(* IEC 61131-3 sources: elnaProjects/ElpcLogic/PomarKc7Unchanged/build_USO_ecl (part 4) *)

  IF getSdvig THEN StrSw.sdvig:= TRUE; END_IF;

  sdvigReset(IN:=StrSw.sdvig, PT:=T#15S);

  IF sdvigReset.Q THEN StrSw.sdvig:=FALSE; END_IF;

  lastOnStatus := StrSw.onStatus;

  (* ---- Распаковка команды ---- *)
  _sunpackerCommand(command := StrSw.inCommand);
  	cmd := _sunpackerCommand.cmd;
  	source := _sunpackerCommand.source;

  (* ---- Обработка команды ---- *)
  IF cmd <> 0 AND lastCmd <> cmd and (((NOT StrSw.opcCommandsDisabled) AND source > 0) OR source = 0) then
  	CASE BYTE_TO_INT(cmd) OF
  	(*cmd_open*) 1 :
  			IF  StrSw.ISVALIDREF_cmdOn THEN StrSw.CmdOn := TRUE;
  				IF StrSw.ISVALIDREF_cmdOff THEN StrSw.CmdOff := FALSE; END_IF;
  			ELSIF  StrSw.ISVALIDREF_cmdOff THEN StrSw.CmdOff := FALSE;  END_IF;
                                lastCmd := cmd;
  			errorCMDTimer(IN := false);
  			_commandErrorTimer := true;
  			StrSw.lastCmdIsOn := true;
  	(*cmd_close*) 2 :
  			IF StrSw.ISVALIDREF_cmdOff THEN StrSw.CmdOff := TRUE;
  				IF StrSw.ISVALIDREF_cmdOn THEN StrSw.CmdOn := FALSE; END_IF;
  			ELSIF StrSw.ISVALIDREF_cmdOn THEN StrSw.CmdOn := FALSE; END_IF;
                                lastCmd := cmd;
  			errorCMDTimer(IN := false);
  			_commandErrorTimer := true;
  			StrSw.lastCmdIsOn := false;
  	(*cmd_reset*) 3 :    IF StrSw.ISVALIDREF_statOn OR StrSw.ISVALIDREF_statOff THEN
  			StrSw.CmdOn := FALSE;
  			StrSw.CmdOff := FALSE;
                                lastCmd :=0;
  			_commandErrorTimer := false;
  			StrSw.lastCmdIsOn := false;
                                 END_IF;
  	END_CASE;
  	source_for_Status := source;
  	cmd_for_Status := cmd;
  	command_error_for_Status := 0;
  END_IF;

  errorCMDTimer(In := _commandErrorTimer, PT :=T#10s);

  (* ---- алгоритм  для команды ВКЛючить ---- *)
  IF (StrSw.onStatus = _statusDualInput.STATUS_ON) and StrSw.lastCmdIsOn then
  	IF StrSw.ISVALIDREF_cmdOn AND StrSw.ISVALIDREF_cmdOff then  StrSw.cmdOn := false; END_IF;

  	 errorCMDTimer(In := false);
  	 _commandErrorTimer := false;
  	 cmd_for_Status := 0;
  	 source_for_Status := 0;
  END_IF;

  (* ---- off ---- *)
  IF (StrSw.onStatus = _statusDualInput.STATUS_OFF) and (NOT StrSw.lastCmdIsOn) then
  	IF StrSw.ISVALIDREF_cmdOn AND StrSw.ISVALIDREF_cmdOff then  StrSw.cmdOff := false; END_IF;

  	 errorCMDTimer(In := false);
  	 _commandErrorTimer := false;
  	 cmd_for_Status := 0;
  	 source_for_Status := 0;
  END_IF;

  (* ---- ошибка исполнения команды ---- *)
  if errorCMDTimer.Q and (cmd_for_Status <> 0) then
  	command_error_for_Status :=  cmd_for_Status;
  	_commandErrorTimer := false;
  	StrSw.CmdOn := false;
  	StrSw.CmdOff := false;
  	lastCmd := 0;
  end_if;

  (* ---- сброс ошибки команды ---- *)
  StrSw.CommandFault := command_error_for_Status <> 0;
  _errorReset(IN := command_error_for_Status <> 0, PT := T#5S);
  IF _errorReset.Q THEN
  	cmd_for_Status := 0;
  	source_for_Status := 0;
  	command_error_for_Status := 0;
  END_IF;

  outputsSets(in := (StrSw.ISVALIDREF_cmdOn and StrSw.cmdOn ) OR (StrSw.ISVALIDREF_cmdOff and StrSw.cmdOff), PT := T#2S);
  	IF NOT outputsSets.Q THEN
  		StrSw.BreakCmdOn := inBreakCmdOn._inversed AND
                      inBreakCmdOn.reliability AND StrSw.ISVALIDREF_inBreakCmdOn;

  		StrSw.BreakCmdOff := inBreakCmdOff._inversed
                      AND inBreakCmdOff.reliability AND StrSw.ISVALIDREF_inBreakCmdOff;
  	END_IF;

  cmdOn := StrSw.cmdOn;
  cmdOff:= StrSw.cmdOff;

  (* ---- формирование зашифрованного статуса для АРМа ---- *)
  StrSw.status := shl(BYTE_TO_DWORD(source_for_Status), 29)
  		OR shl(BYTE_TO_DWORD(cmd_for_Status), 26)
  		OR shl(BYTE_TO_DWORD(command_error_for_Status), 23)
  		OR shl(bool_to_DWORD(StrSw.sdvig), 22)
  		OR shl(bool_to_DWORD(StrSw.OpcCommandsDisabled), 21)
                      OR shl(bool_to_DWORD(StrSw.lastCmdIsOn), 14)
                      OR shl(BOOL_TO_DWORD(StrSw.BreakCmdOff), 13)
  		OR shl(BOOL_TO_DWORD(StrSw.BreakCmdOn), 12)
  		OR shl(BOOL_TO_DWORD(StrSw.ErrorBlock), 11)
  		OR shl(BOOL_TO_DWORD(StrSw.ErrorPowerOff), 10)
  		OR shl(BOOL_TO_DWORD(StrSw.Manual), 8)
  		OR shl(BOOL_TO_DWORD(StrSw.Auto), 7)
  		OR shl(BOOL_TO_DWORD(StrSw.Distance), 6)
  		OR shl(BOOL_TO_DWORD(StrSw.Local), 5)
  		OR shl(BOOL_TO_DWORD(StrSw.Ns), 4)
                  	OR shl(BOOL_TO_DWORD(StrSw.Accident ),3)
  		OR BYTE_TO_DWORD(StrSw.onStatus);
END_FUNCTION_BLOCK

FUNCTION_BLOCK fb_SectionSwitch
  VAR_INPUT
    statOn : BOOL;
    statOff : BOOL;
    statOn_reliability : BOOL;
    statOff_reliability : BOOL;
  END_VAR
  VAR_IN_OUT
    StrSw : struct_SectionSwitch;
  END_VAR
  VAR_INPUT
    basketRolledIn : TYPE_ReliableBit;
    basketRolledOut : TYPE_ReliableBit;
    basketTest : TYPE_ReliableBit;
    inNs : TYPE_ReliableBit;
    inoffKNA : TYPE_ReliableBit;
    inAccident : TYPE_ReliableBit;
    inLocal : TYPE_ReliableBit;
    inDistance : TYPE_ReliableBit;
    inBreakCmdOn : TYPE_ReliableBit;
    inBreakCmdOff : TYPE_ReliableBit;
  END_VAR
  VAR
    onInit : BOOL := FALSE;
    _statOn : BOOL;
    _statOff : BOOL;
    getSdvig : BOOL;
    lastOnStatus : BYTE;
    cmd : BYTE;
    source : BYTE;
    lastCmd : BYTE;
    source_for_Status : BYTE;
    cmd_for_Status : BYTE;
    command_error_for_Status : BYTE;
    _basketRolledIn : TYPE_ReliableBit;
    _basketRolledOut : TYPE_ReliableBit;
    _basketTest : TYPE_ReliableBit;
    _sunpackerCommand : fb_sunpackerCommand;
    _statusDualInput : TYPE_statusDualInput;
    _statusBasket : TYPE_basketStats;
    _commandDualInput : TYPE_commandDualInput;
    _commandErrorTimer : BOOL;
    resetErrorTimer : BOOL;
    _changWithoutCommand : BOOL;
    errorCMDTimer : TON;
    _errorReset : TON;
    sdvigReset : TON;
    outputsSets : TOF;
  END_VAR
  VAR_IN_OUT
    cmdOn : BOOL;
    cmdOff : BOOL;
  END_VAR

  IF NOT onInit THEN
  IF StrSw.ISVALIDREF_cmdOn XOR StrSw.ISVALIDREF_cmdOff THEN
  	IF 	StrSw.ISVALIDREF_cmdOn THEN
  		lastCmd:= 2; (*baseCmdOff*)
  	ELSE
  		lastCmd:= 1; (*baseCmdOn*)
  	END_IF;
  END_IF;
  onInit:=TRUE;
  END_IF;

  (* ---- Формирование состояния тележки ---- *)

  IF (NOT StrSw.ISVALIDREF_basketRolledIn) AND (NOT StrSw.ISVALIDREF_basketRolledOut) THEN
            StrSw.basketStatus:=_statusBasket.BASKET_NOTDEFINED;
  ELSE
  		IF StrSw.ISVALIDREF_basketTest THEN
  		_basketTest:=basketTest;
  	ELSE
  		_basketTest.reliability:=TRUE;
  		_basketTest.value :=FALSE;
  	END_IF;

  	IF StrSw.ISVALIDREF_basketRolledIn THEN
  		_basketRolledIn:=basketRolledIn;
  	ELSE
  		_basketRolledIn:=basketRolledOut;
  		IF StrSw.ISVALIDREF_basketTest THEN
  		_basketRolledIn.value:=NOT (_basketRolledIn.value OR _basketTest.value);
  		ELSE
  		_basketRolledIn.value:= NOT _basketRolledIn.value;
  		END_IF;

  	END_IF;

  	IF StrSw.ISVALIDREF_basketRolledOut THEN
  		_basketRolledOut:=basketRolledOut;
  	ELSE
  		_basketRolledOut:=basketRolledIn;
  		IF StrSw.ISVALIDREF_basketTest THEN
  		_basketRolledOut.value:= NOT (_basketRolledOut.value OR _basketTest.value );
  		ELSE
  			_basketRolledOut.value := NOT _basketRolledout.value;
  		END_IF;

  	END_IF;

  IF _basketRolledIn.reliability AND _basketRolledOut.reliability AND _basketTest.reliability THEN
  		IF (BOOL_TO_INT(_basketRolledIn.value)+BOOL_TO_INT(_basketRolledOut.value)+BOOL_TO_INT(_basketTest.value))=1 THEN
  			IF _basketRolledIn.value THEN
  				StrSw.basketStatus:=_statusBasket.BASKET_ROLLEDIN;
  			ELSIF _basketRolledOut.value THEN
  				StrSw.basketStatus:=_statusBasket.BASKET_ROLLEDOUT;
  			ELSIF _basketTest.value THEN
  				StrSw.basketStatus:=_statusBasket.BASKET_TEST;
  			END_IF;
  		ELSE
  			StrSw.basketStatus:=_statusBasket.BASKET_ERROR;
  		END_IF;
  	ELSE
  		StrSw.basketStatus:=_statusBasket.BASKET_NOTDEFINED;
  	END_IF;
  END_IF;

  (* ---- Если управление с ВУ заблокировано, то в ИМ передаем команду из алгоритма ---- *)
  IF StrSw.inOpcCommandsDisabled THEN
  	StrSw.inCommand := StrSw.inCommand_Alg;
  ELSE (* иначе передаем команду с АРМа*)
  	StrSw.inCommand := StrSw.inCommand_ARM;
  END_IF;

  (* ---- Формирование состояния механизма ---- *)

  IF (StrSw.ISVALIDREF_statOn) OR (StrSw.ISVALIDREF_statOff) THEN
  	IF (StrSw.ISVALIDREF_statOn) AND (StrSw.ISVALIDREF_statOff) THEN
  	StrSw.reliability:= statOn_reliability AND statOff_reliability;
  		_statOn  := statOn;
  		_statOff := statOff;
  	ELSIF (StrSw.ISVALIDREF_statOn) THEN
                       StrSw.reliability:= statOn_reliability;
  		_statOn  := statOn;
  		_statOff := NOT statOn;
  	ELSIF (StrSw.ISVALIDREF_statOff) THEN
  		 StrSw.reliability:= statOff_reliability;
  		_statOn  := NOT statOff;
  		_statOff :=statOff;
  	END_IF;

  	IF StrSw.reliability THEN
  		IF _statOn AND NOT _statOff 		THEN 	StrSw.onStatus := _statusDualInput.STATUS_ON;
  		ELSIF _statOff AND NOT _statOn 	THEN 	StrSw.onStatus := _statusDualInput.Status_OFF;
  		ELSIF NOT _statOn AND NOT _statOff 	THEN 	StrSw.onStatus := _statusDualInput.STATUS_TRANSITIONAL;
  		ELSE					StrSw.onStatus := _statusDualInput.STATUS_ERROR;
                      END_IF;

  	ELSE
  		StrSw.onStatus := _statusDualInput.STATUS_NOTDEFINED;

  	END_IF;
  ELSE
  	CASE BYTE_TO_INT(lastCmd) OF
  		(*baseCmdOn*) 1: StrSw.onStatus  := _statusDualInput.STATUS_ON;
  		(*baseCmdOff*) 2: StrSw.onStatus  := _statusDualInput.STATUS_OFF;

  	ELSE
  		 StrSw.onStatus := _statusDualInput.STATUS_NOTDEFINED;

  	END_CASE;
  END_IF;

  StrSw.Accident := inAccident.value AND inAccident.reliability;
  StrSw.Ns := inNs.value AND inNs.reliability;
  StrSw.Local := inLocal.value AND inLocal.reliability;
  StrSw.Distance := inDistance.value AND inDistance.reliability;
  StrSw.OpcCommandsDisabled := StrSw.inOpcCommandsDisabled;
  StrSw.offKNA := inoffKNA.value AND inoffKNA.reliability;

  (* ---- Формирование признака сдвига ---- *)

  getSdvig := FALSE;
  IF (StrSw.ISVALIDREF_cmdOn OR StrSw.ISVALIDREF_cmdOff) AND NOT StrSw.Local THEN
  	IF NOT (StrSw.CmdOn OR StrSw.CmdOff) THEN
                       IF (lastOnStatus <> StrSw.onStatus AND
  		(StrSw.onStatus <> _statusDualInput.STATUS_NOTDEFINED AND
                       StrSw.onStatus <> _statusDualInput.STATUS_ERROR)     AND
  		(lastOnStatus <> _statusDualInput.STATUS_NOTDEFINED   AND
                       lastOnStatus <> _statusDualInput.STATUS_ERROR))
                      THEN
  			getSdvig   := TRUE;
  		END_IF;
  	END_IF;
  END_IF;

  IF getSdvig THEN StrSw.sdvig:= TRUE; END_IF;

  sdvigReset(IN:=StrSw.sdvig, PT:=T#15S);

  IF sdvigReset.Q THEN StrSw.sdvig:=FALSE; END_IF;

  lastOnStatus := StrSw.onStatus;

  (* ---- Распаковка команды ---- *)
  _sunpackerCommand(command := StrSw.inCommand);
  	cmd := _sunpackerCommand.cmd;
  	source := _sunpackerCommand.source;

  (* ---- Обработка команды ---- *)
  IF cmd <> 0 AND lastCmd <> cmd and (((NOT StrSw.opcCommandsDisabled) AND source > 0) OR source = 0) then
  	CASE BYTE_TO_INT(cmd) OF
  	(*cmd_open*) 1 :
  			IF  StrSw.ISVALIDREF_cmdOn THEN StrSw.CmdOn := TRUE;
  				IF StrSw.ISVALIDREF_cmdOff THEN StrSw.CmdOff := FALSE; END_IF;
  			ELSIF  StrSw.ISVALIDREF_cmdOff THEN StrSw.CmdOff := FALSE;  END_IF;
  			errorCMDTimer(IN := false);
  			_commandErrorTimer := true;
  			StrSw.lastCmdIsOn := true;
  	(*cmd_close*) 2 :
  			IF StrSw.ISVALIDREF_cmdOff THEN StrSw.CmdOff := TRUE;
  				IF StrSw.ISVALIDREF_cmdOn THEN StrSw.CmdOn := FALSE; END_IF;
  			ELSIF StrSw.ISVALIDREF_cmdOn THEN StrSw.CmdOn := FALSE; END_IF;
  			errorCMDTimer(IN := false);
  			_commandErrorTimer := true;
  			StrSw.lastCmdIsOn := false;
  	(*cmd_reset*) 3 :    IF StrSw.ISVALIDREF_statOn OR StrSw.ISVALIDREF_statOff THEN
  			StrSw.CmdOn := FALSE;
  			StrSw.CmdOff := FALSE;
                                lastCmd := 0;
  			_commandErrorTimer := false;
  			StrSw.lastCmdIsOn := false;
                                 END_IF;
  	END_CASE;
  	source_for_Status := source;
  	cmd_for_Status := cmd;
  	command_error_for_Status := 0;
  END_IF;
  lastCmd := cmd;

  errorCMDTimer(In := _commandErrorTimer, PT :=T#10s);

  (* ---- алгоритм  для команды ВКЛючить ---- *)
  IF (StrSw.onStatus = _statusDualInput.STATUS_ON) and (StrSw.lastCmdIsOn) then
  	IF StrSw.ISVALIDREF_cmdOn AND StrSw.ISVALIDREF_cmdOff then  StrSw.cmdOn := false; END_IF;

  	 errorCMDTimer(In := false);
  	 _commandErrorTimer := false;
  	 cmd_for_Status := 0;
  	 source_for_Status := 0;
  END_IF;

  (* ---- off ---- *)
  IF (StrSw.onStatus = _statusDualInput.STATUS_OFF) and (NOT StrSw.lastCmdIsOn) then
  	IF StrSw.ISVALIDREF_cmdOn AND StrSw.ISVALIDREF_cmdOff then  StrSw.cmdOff := false; END_IF;

  	 errorCMDTimer(In := false);
  	 _commandErrorTimer := false;
  	 cmd_for_Status := 0;
  	 source_for_Status := 0;
  END_IF;

  (* ---- ошибка исполнения команды ---- *)
  if errorCMDTimer.Q and (cmd_for_Status <> 0) then
  	command_error_for_Status :=  cmd_for_Status;
  	_commandErrorTimer := false;
  	StrSw.CmdOn := false;
  	StrSw.CmdOff := false;
  	lastCmd := 0;
  end_if;

  (* ---- сброс ошибки команды ---- *)
  StrSw.CommandFault := command_error_for_Status <> 0;
  _errorReset(IN := command_error_for_Status <> 0, PT := T#5S);
  IF _errorReset.Q THEN
  	cmd_for_Status := 0;
  	source_for_Status := 0;
  	command_error_for_Status := 0;
  END_IF;

  outputsSets(in := (StrSw.ISVALIDREF_cmdOn and StrSw.cmdOn ) OR (StrSw.ISVALIDREF_cmdOff and StrSw.cmdOff), PT := T#2S);
  	IF NOT outputsSets.Q THEN
  		StrSw.BreakCmdOn := inBreakCmdOn._inversed AND inBreakCmdOn.reliability AND StrSw.ISVALIDREF_inBreakCmdOn;
  		StrSw.BreakCmdOff := inBreakCmdOff._inversed AND inBreakCmdOff.reliability AND StrSw.ISVALIDREF_inBreakCmdOff;
  	END_IF;

  cmdOn := StrSw.cmdOn;
  cmdOff:= StrSw.cmdOff;

  (* ---- формирование зашифрованного статуса для АРМа ---- *)
  StrSw.status := shl(BYTE_TO_DWORD(source_for_Status), 29)
  		OR shl(BYTE_TO_DWORD(cmd_for_Status), 26)
  		OR shl(BYTE_TO_DWORD(command_error_for_Status), 23)
  		OR shl(bool_to_DWORD(StrSw.sdvig), 22)
  		OR shl(bool_to_DWORD(StrSw.OpcCommandsDisabled), 21)
                      OR shl(BOOL_TO_DWORD(StrSw.offKNA), 17)
                      OR shl(bool_to_DWORD(StrSw.lastCmdIsOn), 14)
                      OR shl(BOOL_TO_DWORD(StrSw.BreakCmdOff), 13)
  		OR shl(BOOL_TO_DWORD(StrSw.BreakCmdOn), 12)
                      OR shl(BYTE_TO_DWORD(StrSw.basketStatus), 8)
  		OR shl(BOOL_TO_DWORD(StrSw.Distance), 6)
  		OR shl(BOOL_TO_DWORD(StrSw.Local), 5)
  		OR shl(BOOL_TO_DWORD(StrSw.Ns), 4)
                  	OR shl(BOOL_TO_DWORD(StrSw.Accident ),3)
  		OR BYTE_TO_DWORD(StrSw.onStatus);
END_FUNCTION_BLOCK

FUNCTION_BLOCK fb_meandr
  VAR
    _output : BOOL;
  END_VAR
  VAR_INPUT
    period : TIME := T#300MS;
  END_VAR
  VAR
    timer : TON;
    FALSE_val : BOOL := FALSE;
    TRUE_val : BOOL := TRUE;
  END_VAR
  VAR_IN_OUT
    output : BOOL;
  END_VAR

  timer(in:=NOT FALSE_val,PT:=period);

  IF timer.Q THEN
      _output:=_output XOR TRUE_val;
      timer(in:=FALSE);
  END_IF;

  output:=_output;
END_FUNCTION_BLOCK

FUNCTION_BLOCK fb_singleSignal
  VAR_INPUT
    signal : TYPE_ReliableBit;
  END_VAR
  VAR_IN_OUT
    str_SS : struct_singleSignal;
  END_VAR
  VAR
    TimerOn : TON;
    TimerOff : TOF;
  END_VAR

  str_SS.reliability:=signal.reliability;

  IF NOT str_SS.inverse THEN
  TimerOn(IN:=(signal.value AND str_SS.reliability AND NOT str_SS.Disabled_Sig), PT:=str_SS.DelayOn);
  ELSE
  TimerOn(IN:=(signal._inversed AND str_SS.reliability AND NOT str_SS.Disabled_Sig), PT:=str_SS.DelayOn);
  END_IF;

  TimerOff(IN:=TimerOn.Q, PT:=str_SS.DelayOff);

  str_SS.Q:=TimerOff.Q;

  str_SS.status:= SHL(BOOL_TO_DWORD(NOT str_SS.reliability), 15)
  	OR BOOL_TO_DWORD(str_SS.Q);
END_FUNCTION_BLOCK

FUNCTION_BLOCK fb_singleOutput
  VAR_IN_OUT
    signal : BOOL;
    str_SO : struct_singleOutput;
  END_VAR
  VAR
    pulseTimer : TON;
    resetCmdTimer : TON;
    TON_Command : TON;
    source : BYTE;
    cmd : BYTE;
    lastCmd : BYTE;
    source_for_Status : BYTE;
    cmd_for_Status : BYTE;
    command_error_for_Status : BYTE;
    pulseTimerPriznak : BOOL;
    resetCmdTimerPriznak : BOOL;
    _sunpackerCommand : fb_sunpackerCommand;
  END_VAR

  str_SO.OpcCommandsDisabled := str_SO.inOpcCommandsDisabled;

  (* ---- Если управление с ВУ заблокировано, то передаем команду из алгоритма ---- *)
  IF str_SO.inOpcCommandsDisabled THEN
  	str_SO.inCommand := str_SO.inCommand_Alg;
  ELSE (* иначе передаем команду с АРМа*)
  	str_SO.inCommand := str_SO.inCommand_ARM;
  END_IF;

  (*Распаковка команды*)
  _sunpackerCommand(command := str_SO.inCommand);
  	cmd := _sunpackerCommand.cmd;
  	source := _sunpackerCommand.source;

  (*Обработка команды*)
  IF cmd <> 0 AND lastCmd <> cmd and (((NOT str_SO.OpcCommandsDisabled) AND source > 0) OR source = 0) then
  	CASE BYTE_TO_INT(cmd) OF
  	(*cmd_on*) 1 :
  			str_SO.Q := TRUE;
  			pulseTimer(IN := FALSE);
  			pulseTimerPriznak := FALSE;
  			resetCmdTimer(IN := FALSE);
  			resetCmdTimerPriznak := TRUE;
  	(*cmd_off*) 2 :
  			str_SO.Q := FALSE;
  			pulseTimer(IN := FALSE);
  			pulseTimerPriznak := FALSE;
  			resetCmdTimer(IN := FALSE);
  			resetCmdTimerPriznak := TRUE;
  	(*cmd_pulse*) 3 :
  			str_SO.Q := TRUE;
                                pulseTimer(IN := FALSE);
                                pulseTimerPriznak := TRUE;
  			resetCmdTimer(IN := FALSE);
                                resetCmdTimerPriznak := FALSE;
  	END_CASE;
  	source_for_Status := source;
  	cmd_for_Status := cmd;
  	command_error_for_Status := 0;
  END_IF;
  lastCmd := cmd;

  pulseTimer(IN := pulseTimerPriznak, PT := str_SO.wait_time);
  pulseTimer();
  IF pulseTimer.Q THEN
  	pulseTimer(IN := FALSE);
  	pulseTimerPriznak := FALSE;

  	str_SO.Q := FALSE;

  	source_for_Status := 0;
  	cmd_for_Status := 0;
  	command_error_for_Status := 0;
  END_IF;

  resetCmdTimer(IN := resetCmdTimerPriznak, PT := T#10S);
  resetCmdTimer();
  IF resetCmdTimer.Q THEN
  	resetCmdTimer(IN := FALSE);
  	resetCmdTimerPriznak := FALSE;

  	source_for_Status := 0;
  	cmd_for_Status := 0;
  	command_error_for_Status := 0;
  END_IF;

  signal:= str_SO.Q;

  (*TON_Command(IN:= (inCommand <> 0) AND (source = 0), PT:= T#2S);*)
      (*IF TON_Command.Q THEN*)
          (*inCommand := 0;*)
      (*END_IF;*)
  str_SO.status :=                           shl(BYTE_TO_DWORD(source_for_Status), 29)
  				OR shl(BYTE_TO_DWORD(cmd_for_Status), 26)
  				OR shl(BYTE_TO_DWORD(command_error_for_Status), 23)
  				OR shl(BOOL_TO_DWORD(str_SO.OpcCommandsDisabled), 21)
  				OR BOOL_TO_DWORD(str_SO.Q);
END_FUNCTION_BLOCK

FUNCTION_BLOCK fb_DiscretParametr
  VAR_IN_OUT
    StrDP : struct_DiscretParametr;
  END_VAR
  VAR
    _sunpackerCommand : fb_sunpackerCommand;
    source : BYTE;
    cmd : BYTE;
    parametr : BYTE;
    lastParametr : BYTE;
    source_for_Status : BYTE;
    cmd_for_Status : BYTE;
    command_error_for_Status : BYTE;
    resetCmdTimer : TON;
    resetCmdTimerPriznak : BOOL;
    secondTact : BOOL;
  END_VAR

  IF NOT secondTact THEN
  	StrDP.Value := StrDP.currentValue;
  	secondTact := true;
  END_IF;

  StrDP.OpcCommandsDisabled := StrDP.inOpcCommandsDisabled;

  (* ---- Если управление с ВУ заблокировано, то передаем команду из алгоритма ---- *)
  IF StrDP.inOpcCommandsDisabled THEN
  	StrDP.inCommand := StrDP.inCommand_Alg;
  ELSE (* иначе передаем команду с АРМа*)
  	StrDP.inCommand := StrDP.inCommand_ARM;
  END_IF;

  _sunpackerCommand(command := StrDP.inCommand);
  	source := _sunpackerCommand.source;
            parametr := _sunpackerCommand.parametr;
  	cmd := _sunpackerCommand.cmd;

  IF NOT StrDP.inOpcCommandsDisabled THEN
  StrDP.newValue:= BYTE_TO_UINT(parametr);
  END_IF;

  IF cmd <> 0 AND StrDP.Value <> StrDP.newValue AND (((NOT StrDP.opcCommandsDisabled) AND source > 0) OR source = 0) then
  	CASE BYTE_TO_INT(cmd) OF
  	(*cmd_ChangeValue*) 1 :
                                    StrDP.Value := StrDP.newValue;
                                    StrDP.opcCommandsDisabled:=FALSE;
  	END_CASE;
  	source_for_Status := source;
  	cmd_for_Status := cmd;
  	resetCmdTimer(IN := FALSE);
  	resetCmdTimerPriznak := TRUE;
  END_IF;

  lastParametr := parametr;

  StrDP.status := SHL(BYTE_TO_DWORD(source_for_Status), 29)
  			OR SHL(BYTE_TO_DWORD(cmd_for_Status), 26)
  			OR SHL(BYTE_TO_DWORD(command_error_for_Status), 23)
  			OR SHL(BOOL_TO_DWORD(StrDP.OpcCommandsDisabled ), 21)
                                OR SHL(UINT_TO_DWORD(StrDP.Value), 5);

  resetCmdTimer(IN := resetCmdTimerPriznak, PT := T#5S);
  IF resetCmdTimer.Q THEN
  	resetCmdTimerPriznak := FALSE;
  	source_for_Status := 0;
  	cmd_for_Status := 0;
  	command_error_for_Status := 0;
  END_IF;
END_FUNCTION_BLOCK

FUNCTION_BLOCK fb_AnalogParametr
  VAR_IN_OUT
    StrAP : struct_AnalogParametr;
  END_VAR
  VAR
    _sunpackerCommand : fb_sunpackerCommand;
    source : BYTE;
    cmd : BYTE;
    source_for_Status : BYTE;
    cmd_for_Status : BYTE;
    command_error_for_Status : BYTE;
    resetCmdTimer : TON;
    resetCmdTimerPriznak : BOOL;
    secondTact : BOOL;
    inp : LREAL;
    rABS : LREAL;
  END_VAR

  IF NOT secondTact THEN
  	StrAP.Value := StrAP.currentValue;
  	secondTact := true;
  END_IF;

  StrAP.OpcCommandsDisabled := StrAP.inOpcCommandsDisabled;

   (* ---- Если управление с ВУ заблокировано, то передаем команду из алгоритма ---- *)
  IF StrAP.inOpcCommandsDisabled THEN
  	StrAP.inCommand := StrAP.inCommand_Alg;
  ELSE (* иначе передаем команду с АРМа*)
  	StrAP.inCommand := StrAP.inCommand_ARM;
  END_IF;

  _sunpackerCommand(command := StrAP.inCommand);
  	source := _sunpackerCommand.source;
  	cmd := _sunpackerCommand.cmd;

  IF cmd <> 0 AND StrAP.newValue <> StrAP.Value and (((NOT StrAP.opcCommandsDisabled) AND source > 0) OR source = 0) then
  	CASE BYTE_TO_INT(cmd) OF
  	(*cmd_ChangeValue*) 1 :
  				StrAP.isValidValue := TRUE;
  				IF StrAP.minVal_ISVALIDREF AND StrAP.isValidValue THEN
  					IF StrAP.newValue < StrAP.minVal THEN
  						StrAP.isValidValue := FALSE;
  					END_IF;
  				END_IF;
  				IF StrAP.maxVal_ISVALIDREF AND StrAP.isValidValue THEN
  					IF StrAP.newValue > StrAP.maxVal THEN
  						StrAP.isValidValue := FALSE;
  					END_IF;
  				END_IF;
  				IF StrAP.maxStep_ISVALIDREF AND StrAP.isValidValue  THEN
  					inp := StrAP.Value - StrAP.newValue;
  					IF inp < 0.0 THEN
  						rABS := -inp;
  					ELSE
  						rABS := inp;
  					END_IF;
  					IF rABS > StrAP.maxStep THEN
  						StrAP.isValidValue := FALSE;
  					END_IF;
  				END_IF;
  				IF StrAP.isValidValue THEN
  					StrAP.Value := StrAP.newValue;
  					command_error_for_Status := 0;
  				ELSE
  					command_error_for_Status := cmd;
  				END_IF;
  	END_CASE;
  	source_for_Status := source;
  	cmd_for_Status := cmd;
  	resetCmdTimer(IN := FALSE);
  	resetCmdTimerPriznak := TRUE;
  END_IF;

  resetCmdTimer(IN := resetCmdTimerPriznak, PT := T#5S);
  IF resetCmdTimer.Q THEN
  	resetCmdTimerPriznak := FALSE;
  	source_for_Status := 0;
  	cmd_for_Status := 0;
  	command_error_for_Status := 0;
  END_IF;

  StrAP.status := SHL(BYTE_TO_DWORD(source_for_Status), 29)
  			OR SHL(BYTE_TO_DWORD(cmd_for_Status), 26)
  			OR SHL(BYTE_TO_DWORD(command_error_for_Status), 23)
  			OR SHL(BOOL_TO_DWORD(StrAP.OpcCommandsDisabled ), 21);
END_FUNCTION_BLOCK

FUNCTION_BLOCK proc_IM
  VAR
    fb_Kran1 : fb_Kran;
    fb_Kran2 : fb_Kran;
    fb_Kran3b : fb_Kran;
    fb_Kran4 : fb_Kran;
    fb_Kran5 : fb_Kran;
    fb_Kran6 : fb_Kran;
    fb_nu1 : fb_OilPump;
    fb_nu2 : fb_OilPump;
    fb_pns : fb_Switch;
    fb_v1_Avom : fb_Switch;
    fb_v2_Avom : fb_Switch;
    fb_Ten : fb_Switch;
    fb_mv : fb_SectionSwitch;
    fb_PLC_Control : fb_meandr;
  END_VAR
  VAR_EXTERNAL
    di : DiConfig;
    od : DOconfig;
    IM : ImConfig;
  END_VAR
  VAR
    fb_KZ_10kv : fb_singleSignal;
    fb_OsevoiSdvig_pravo : fb_singleSignal;
    fb_OsevoiSdvig_levo : fb_singleSignal;
    fb_dP_oilgaz_low : fb_singleSignal;
    fb_P_oil_low : fb_singleSignal;
    fb_dP_gazgaz_Kran1 : fb_singleSignal;
    fb_Vozb_ProboiVentila : fb_singleSignal;
    fb_Vozb_AsinchHod : fb_singleSignal;
    fb_Vozb_ReSynchronize : fb_singleSignal;
    fb_Vozb_ControlVozbuditela : fb_singleSignal;
    fb_NS_ForsingVozbugdenia : fb_singleSignal;
    fb_NS_Vozbyditela : fb_singleSignal;
    fb_Vozb_AVR_off : fb_singleSignal;
    fb_Vozb_AutoUprVozbuditela_off : fb_singleSignal;
    fb_Vozb_KontaktorON : fb_singleSignal;
    fb_Vozb_Overload : fb_singleSignal;
    fb_AO_KC : fb_singleSignal;
    fb_AOGPA_PRU : fb_singleSignal;
    fb_BEO_Ready : fb_singleSignal;
    fb_BEO_Srabat : fb_singleSignal;
    fb_BEO_ON_knopkaSHU : fb_singleSignal;
    fb_BEO_ON_knopkaPRU : fb_singleSignal;
    fb_NOGPA_knopkaSHU : fb_singleSignal;
    fb_AOGPA_knopkaSHU : fb_singleSignal;
    fb_DverShkafaOtkryta : fb_singleSignal;
    fb_QF1_on : fb_singleSignal;
    fb_QF2_on : fb_singleSignal;
    fb_QF23_on : fb_singleSignal;
    fb_QF4_QF5_on : fb_singleSignal;
    fb_QF6_QF7_on : fb_singleSignal;
    fb_QF8_QF9_on : fb_singleSignal;
    fb_QF10_QF11_on : fb_singleSignal;
    fb_QF12_QF13_on : fb_singleSignal;
    fb_QF14_QF15_on : fb_singleSignal;
    fb_QF22_on : fb_singleSignal;
    fb_NS_G1_G2 : fb_singleSignal;
    fb_NS_G3_G4 : fb_singleSignal;
    fb_NS_G15_G16 : fb_singleSignal;
    fb_NS_G17 : fb_singleSignal;
    fb_NS_G5_G6 : fb_singleSignal;
    fb_NS_G7_G8 : fb_singleSignal;
    fb_NS_G18_G19 : fb_singleSignal;
    fb_NS_G10_G11 : fb_singleSignal;
    fb_NS_G13_G14 : fb_singleSignal;
    fb_Lampa_NO : fb_singleOutput;
    fb_VzvodBREO : fb_singleOutput;
    fb_AO_GPA : fb_singleOutput;
    fb_SbrosBREO : fb_singleOutput;
    fb_IndikicijaPS_fonar : fb_singleOutput;
    fb_IndikicijaAS_fonar : fb_singleOutput;
    fb_mv_off_KNA : fb_singleOutput;
    fb_TypeSwitch : fb_DiscretParametr;
    fb_AutoNU_mainNU : fb_DiscretParametr;
    fb_AutoNU_Reset_HasNU : fb_DiscretParametr;
    fb_AutoAvom_hysteresis : fb_AnalogParametr;
    fb_AutoAvom_onTemp1 : fb_AnalogParametr;
    fb_AutoAvom_onTemp2 : fb_AnalogParametr;
    fb_AutoPns_UstRun : fb_AnalogParametr;
    fb_AutoPns_UstStop : fb_AnalogParametr;
    fb_PuskOilSystem_UstdPmg : fb_AnalogParametr;
    fb_AutoTen_offTemperature : fb_AnalogParametr;
    fb_AutoNU_Ust_Swap : fb_AnalogParametr;
    fb_testdPmg_Ust_dPLow : fb_AnalogParametr;
    fb_AntiPompag_UgolVNA : fb_AnalogParametr;
    fb_AntiPompag_K : fb_AnalogParametr;
    fb_AntiPompag_A : fb_AnalogParametr;
    fb_AntiPompag_y0 : fb_AnalogParametr;
  END_VAR

  (* Циклический опрос. ИМ *)

  (* GPIO *)
  fb_PLC_Control(output:=od.gpio_out.bits[0]);

  (* Кран 1 *)
  fb_Kran1(statOn := di.di_0.bits[0]._inversed, statOn_reliability:= di.di_0.bits[0].reliability,
           statOff := di.di_0.bits[1]._inversed, statOff_reliability:= di.di_0.bits[1].reliability,
           inSo := di.di_12.bits[0], inSz := di.di_12.bits[1],
           inDp:= di.di_2.bits[0],
           cmdOn:=od.do_0.bits[0], cmdOff:=od.do_0.bits[1],
           strKr:= IM.Kran1  );

  (* Кран 2 *)
  fb_Kran2(statOn := di.di_0.bits[2]._inversed, statOn_reliability:= di.di_0.bits[2].reliability,
           statOff := di.di_0.bits[3]._inversed,  statOff_reliability:= di.di_0.bits[3].reliability,
           inSo := di.di_12.bits[2], inSz := di.di_12.bits[3],
           cmdOn:=od.do_0.bits[2], cmdOff:=od.do_0.bits[3],
           strKr:= IM.Kran2  );

  (* Кран 3b *)
  fb_Kran3b(statOn := di.di_0.bits[4]._inversed, statOn_reliability:= di.di_0.bits[4].reliability,
           statOff := di.di_0.bits[5]._inversed,  statOff_reliability:= di.di_0.bits[5].reliability,
           inSo := di.di_12.bits[4], inSz := di.di_12.bits[5],
           cmdOn:=od.do_0.bits[4], cmdOff:=od.do_0.bits[5],
           strKr:= IM.Kran3b  );

  (* Кран 4 *)
  fb_Kran4(statOn := di.di_0.bits[6]._inversed, statOn_reliability:= di.di_0.bits[6].reliability,
           statOff := di.di_0.bits[7]._inversed,  statOff_reliability:= di.di_0.bits[7].reliability,
           inSo := di.di_12.bits[6], inSz := di.di_12.bits[7],
           cmdOn:=od.do_0.bits[6], cmdOff:=od.do_0.bits[7],
           strKr:= IM.Kran4  );

  (* Кран 5 *)
  fb_Kran5(statOn := di.di_1.bits[0]._inversed, statOn_reliability:= di.di_1.bits[0].reliability,
           statOff := di.di_1.bits[1]._inversed,  statOff_reliability:= di.di_1.bits[1].reliability,
           inSo := di.di_13.bits[0], inSz := di.di_13.bits[1],
           cmdOn:=od.do_0.bits[8], cmdOff:=od.do_0.bits[9],
           strKr:= IM.Kran5  );

  (* Кран 6НР *)
  fb_Kran6(statOn := di.di_1.bits[2].value, statOn_reliability:= di.di_1.bits[2].reliability,
           statOff := di.di_1.bits[3].value,  statOff_reliability:= di.di_1.bits[3].reliability,
           cmdOn:=od.do_1.bits[14], cmdOff:=od.do_1.bits[15],
           strKr:= IM.Kran6  );

  (*  НУ1 Насос уплотнения *)
  fb_nu1(statOn := di.di_2.bits[5].value, statOn_reliability:= di.di_2.bits[5].reliability,
           inBreakCmdOn := di.di_10.bits[2],
           cmdOn:=od.do_1.bits[2], cmdOff:=od.do_1.bits[3],
           StrSw:= IM.nu1  );

  (*  НУ2 Насос уплотнения *)
  fb_nu2(statOn := di.di_2.bits[6].value, statOn_reliability:= di.di_2.bits[6].reliability,
           inBreakCmdOn := di.di_10.bits[4],
           cmdOn:=od.do_1.bits[4], cmdOff:=od.do_1.bits[5],
           StrSw:= IM.nu2  );

  (*  ПНС Насос смазки *)
  fb_pns(statOn := di.di_2.bits[7].value, statOn_reliability:= di.di_2.bits[7].reliability,
           inBreakCmdOn := di.di_10.bits[0],
           cmdOn:=od.do_1.bits[0] , cmdOff:=od.do_1.bits[1],
           StrSw:= IM.pns  );

  (*  В1 АВОМ вентилятор охлаждения *)
  fb_v1_Avom(statOn := di.di_3.bits[0].value, statOn_reliability:= di.di_3.bits[0].reliability,
           inBreakCmdOn := di.di_10.bits[6],
           cmdOn:=od.do_1.bits[6] , cmdOff:=od.do_1.bits[7],
           StrSw:= IM.v1_Avom  );

  (*  В2 АВОМ вентилятор охлаждения *)
  fb_v2_Avom(statOn := di.di_3.bits[1].value, statOn_reliability:= di.di_3.bits[1].reliability,
           inBreakCmdOn := di.di_11.bits[0],
           cmdOn:=od.do_1.bits[8] , cmdOff:=od.do_1.bits[9],
           StrSw:= IM.v2_Avom  );

  (*  ТЭН *)
    fb_Ten(statOn := di.di_14.bits[0].value, statOn_reliability:= di.di_14.bits[0].reliability,
           statOff := di.di_14.bits[1].value, statOff_reliability:= di.di_14.bits[1].reliability,
           cmdOn:=od.do_1.bits[13] , cmdOff:=od.do_2.bits[1],
           StrSw:= IM.Ten  );

  (*  МВ масляный выключатель *)
      fb_mv(statOff := di.di_4.bits[7].value, statOff_reliability:= di.di_4.bits[7].reliability,
           inBreakCmdOff := di.di_11.bits[2], inoffKNA:= di.di_5.bits[2],
           basketRolledin:= di.di_5.bits[1], basketRolledout:= di.di_5.bits[0],
           cmdOn:=od.do_1.bits[10] , cmdOff:=od.do_1.bits[11],
           StrSw:= IM.mv  );

  (*************************************************** singleSignals ********************************************)

   (* Перепад давления «газ-газ» на кране 1 ≤1 кгс/см² *)
  fb_dP_gazgaz_Kran1(signal :=di.di_2.bits[0], str_SS := IM.SingleSignals.dP_gazgaz_Kran1);

   (* Осевой сдвиг ротора вправо ≥3,7 кгс/см² *)
  fb_OsevoiSdvig_pravo(signal :=di.di_2.bits[1], str_SS := IM.SingleSignals.OsevoiSdvig_pravo);

   (* Осевой сдвиг ротора влево ≥3,7 кгс/см² *)
  fb_OsevoiSdvig_levo(signal :=di.di_2.bits[2], str_SS := IM.SingleSignals.OsevoiSdvig_levo);

   (* Низкий перепад давления «масло-газ» ≤1 кгс/см² *)
  fb_dP_oilgaz_low(signal :=di.di_2.bits[3], str_SS := IM.SingleSignals.dP_oilgaz_low);

  (* Низкое давление масла смазки ≤ 0,4 кгс/см² *)
  fb_P_oil_low(signal :=di.di_2.bits[4], str_SS := IM.SingleSignals.P_oil_low);

      (* Защита по замыканию на землю 10 кВ (пробой изоляции кабелей) *)
  fb_KZ_10kv(signal :=di.di_3.bits[2], str_SS := IM.SingleSignals.KZ_10kv);

      (* Пробой вентиля *)
  fb_Vozb_ProboiVentila(signal :=di.di_3.bits[3], str_SS := IM.SingleSignals.Vozb_ProboiVentila);

      (* Асинхронный ход и перегрузка *)
  fb_Vozb_AsinchHod(signal :=di.di_3.bits[4], str_SS := IM.SingleSignals.Vozb_AsinchHod);

      (* Работа схемы ресинхронизации *)
  fb_Vozb_ReSynchronize(signal :=di.di_3.bits[5], str_SS := IM.SingleSignals.Vozb_ReSynchronize);

      (* Контроль состояния возбудительного устройства  *)
  fb_Vozb_ControlVozbuditela(signal :=di.di_3.bits[6], str_SS := IM.SingleSignals.Vozb_ControlVozbuditela);

      (* Неисправность форсировки воз-буждения  *)
  fb_NS_ForsingVozbugdenia(signal :=di.di_3.bits[7], str_SS := IM.SingleSignals.NS_ForsingVozbugdenia);

    (* Неисправность возбудительного устройства  *)
  fb_NS_Vozbyditela(signal :=di.di_4.bits[0], str_SS := IM.SingleSignals.NS_Vozbyditela);

    (* Отключен АВР  *)
  fb_Vozb_AVR_off(signal :=di.di_4.bits[1], str_SS := IM.SingleSignals.Vozb_AVR_off);

    (* Отключено автоматическое управление возбудителем  *)
  fb_Vozb_AutoUprVozbuditela_off(signal :=di.di_4.bits[2], str_SS := IM.SingleSignals.Vozb_AutoUprVozbuditela_off);

    (* Контактор возбуждения включен  *)
  fb_Vozb_KontaktorON(signal :=di.di_4.bits[3], str_SS := IM.SingleSignals.Vozb_KontaktorON);

    (* Перегрузка  *)
  fb_Vozb_Overload(signal :=di.di_4.bits[4], str_SS := IM.SingleSignals.Vozb_Overload);

    (* Аварийный останов цеха  *)
  fb_AO_KC(signal :=di.di_5.bits[5], str_SS := IM.SingleSignals.AO_KC);

    (* АО ГПА от кнопки на ПРУ  *)
  fb_AOGPA_PRU(signal :=di.di_5.bits[6], str_SS := IM.SingleSignals.AOGPA_PRU);

    (* Готовность включения БЭО по отказу контроллера  *)
  fb_BEO_Ready(signal :=di.di_6.bits[0], str_SS := IM.SingleSignals.BEO_Ready);

    (* Срабатывание БЭАО  *)
  fb_BEO_Srabat(signal :=di.di_6.bits[1], str_SS := IM.SingleSignals.BEO_Srabat);

    (* Запуск БЭАО от кнопки ЭАО ШУ  *)
  fb_BEO_ON_knopkaSHU(signal :=di.di_6.bits[2], str_SS := IM.SingleSignals.BEO_ON_knopkaSHU);

    (* Экстренный аварийный останов ЭАО ЭГПА с ПРУ   *)
  fb_BEO_ON_knopkaPRU(signal :=di.di_6.bits[7], str_SS := IM.SingleSignals.BEO_ON_knopkaPRU);

    (* НО ГПА от ШУ   *)
  fb_NOGPA_knopkaSHU(signal :=di.di_6.bits[3], str_SS := IM.SingleSignals.NOGPA_knopkaSHU);

    (* АО ГПА от ШУ   *)
  fb_AOGPA_knopkaSHU(signal :=di.di_6.bits[4], str_SS := IM.SingleSignals.AOGPA_knopkaSHU);

    (* Дверь шкафа открыта   *)
  fb_DverShkafaOtkryta(signal :=di.di_6.bits[6], str_SS := IM.SingleSignals.DverShkafaOtkryta);

    (* Выключатель основного ввода питания QF1  в положении включен   *)
  fb_QF1_on(signal :=di.di_7.bits[6], str_SS := IM.SingleSignals.QF1_on);

    (* Выключатель резервного ввода питания QF2  в положении включен   *)
  fb_QF2_on(signal :=di.di_7.bits[7], str_SS := IM.SingleSignals.QF2_on);

    (* Выключатель питания кранов:  QF23 110 В в положении включен   *)
  fb_QF23_on(signal :=di.di_8.bits[0], str_SS := IM.SingleSignals.QF23_on);

    (* Выключатели группы 1: QF4, QF5 в положении включен   *)
  fb_QF4_QF5_on(signal :=di.di_8.bits[1], str_SS := IM.SingleSignals.QF4_QF5_on);

    (* Выключатели группы 2: QF6, QF7 в положении включен   *)
  fb_QF6_QF7_on(signal :=di.di_8.bits[2], str_SS := IM.SingleSignals.QF6_QF7_on);

    (* Выключатели группы 3: QF8, QF9 в положении включен   *)
  fb_QF8_QF9_on(signal :=di.di_8.bits[3], str_SS := IM.SingleSignals.QF8_QF9_on);

    (* Выключатели группы 4: QF10, QF11 в положении включен   *)
  fb_QF10_QF11_on(signal :=di.di_8.bits[4], str_SS := IM.SingleSignals.QF10_QF11_on);

    (* Выключатели группы 5: QF12, QF13 в положении включен   *)
  fb_QF12_QF13_on(signal :=di.di_8.bits[5], str_SS := IM.SingleSignals.QF12_QF13_on);

    (* Выключатели группы 6: QF14, QF15 в положении включен   *)
  fb_QF14_QF15_on(signal :=di.di_8.bits[6], str_SS := IM.SingleSignals.QF14_QF15_on);

    (* Выключатели группы : QF22 в положении включен   *)
  fb_QF22_on(signal :=di.di_14.bits[2], str_SS := IM.SingleSignals.QF22_on);

    (* Неисправность источников питания группы 1: G1, G2 (=24 В)   *)
  fb_NS_G1_G2(signal :=di.di_8.bits[7], str_SS := IM.SingleSignals.NS_G1_G2);

    (* Неисправность источников питания группы 2: G3, G4 (=24 В)   *)
  fb_NS_G3_G4(signal :=di.di_9.bits[0], str_SS := IM.SingleSignals.NS_G3_G4);

    (* Неисправность источников питания внутренних ПТС: G15, G16 (=24 В)   *)
  fb_NS_G15_G16(signal :=di.di_9.bits[1], str_SS := IM.SingleSignals.NS_G15_G16);

    (* Неисправность источника питания аналоговых сигналов: G17 (=24 В)   *)
  fb_NS_G17(signal :=di.di_9.bits[2], str_SS := IM.SingleSignals.NS_G17);

    (* Неисправность источников питания группы 3: G5, G6 (=24 В)   *)
  fb_NS_G5_G6(signal :=di.di_9.bits[3], str_SS := IM.SingleSignals.NS_G5_G6);

    (* Неисправность источников питания группы 4: G7, G8 (=24 В)   *)
  fb_NS_G7_G8(signal :=di.di_9.bits[4], str_SS := IM.SingleSignals.NS_G7_G8);

    (* Неисправность источников питания внешних цепей: G18, G19 (=24 В)   *)
  fb_NS_G18_G19(signal :=di.di_9.bits[5], str_SS := IM.SingleSignals.NS_G18_G19);

    (* Неисправность источников питания группы 5: G9, G10, G11, G12 (=110 В)   *)
  fb_NS_G10_G11(signal :=di.di_9.bits[6], str_SS := IM.SingleSignals.NS_G10_G11);

    (* Неисправность источников питания G13, G14 (=24 В)   *)
  fb_NS_G13_G14(signal :=di.di_9.bits[7], str_SS := IM.SingleSignals.NS_G13_G14);

  (*************************************************** SingleOutputs ********************************************)

  (* Идикация НО (подсветка кнопки на шкафу)   *)
  fb_Lampa_NO(str_SO := IM.SingleOutputs.Lampa_NO, signal:=od.do_2.bits[11]);

  (* Взвод включения БЭАО по неисправности ПТС   *)
  fb_VzvodBREO(str_SO := IM.SingleOutputs.VzvodBREO, signal:=od.do_2.bits[14]);

  (* Авария ЭГПА в КЦ   *)
  fb_AO_GPA(str_SO := IM.SingleOutputs.AO_GPA, signal:=od.do_2.bits[0]);

  (* Сброс включения БЭАО по неисправности ПТС   *)
  fb_SbrosBREO(str_SO := IM.SingleOutputs.SbrosBREO, signal:=od.do_2.bits[15]);

  (* Индикация ПС Фонарь   *)
  fb_IndikicijaPS_fonar(str_SO := IM.SingleOutputs.IndikicijaPS_fonar, signal:=od.do_2.bits[13]);

  (* Индикация АС Фонарь   *)
  fb_IndikicijaAS_fonar(str_SO := IM.SingleOutputs.IndikicijaAS_fonar, signal:=od.do_2.bits[12]);

  (* Отключение МВ1 от КНА   *)
  fb_mv_off_KNA(str_SO := IM.SingleOutputs.mv_off_KNA, signal:=od.do_1.bits[12]);

   (**************************************** Аналоговые и Дискретные параметры ***********************************)

    (* Гистерезис температуры вклюючения вентиляторов в алгоритме АвтоАВОМ  *)
  fb_AutoAvom_hysteresis(StrAP:=IM.AutoAvom_hysteresis);

    (* Температура вклюючения АВОМ1 в алгоритме АвтоАВОМ  *)
  fb_AutoAvom_onTemp1(StrAP:=IM.AutoAvom_onTemp1);

    (* Температура вклюючения АВОМ1 в алгоритме АвтоАВОМ  *)
  fb_AutoAvom_onTemp2(StrAP:=IM.AutoAvom_onTemp2);

    (* Температура включения ПНС в алгоритме АвтоПНС  *)
  fb_AutoPns_UstRun(StrAP:=IM.AutoPns_UstRun);

    (* Температура отключения ПНС в алгоритме АвтоПНС  *)
  fb_AutoPns_UstStop(StrAP:=IM.AutoPns_UstStop);

    (* Давление масло-газ включения защит в алгоритме Пуск Маслосистемы  *)
  fb_PuskOilSystem_UstdPmg(StrAP:=IM.PuskOilSystem_UstdPmg);

  (* Температура отключения ТЭНа в алгоритме АвтоТЭН *)
  fb_AutoTen_offTemperature(StrAP:=IM.AutoTen_offTemperature);

  (* Уставка включения резервного НУ по перепаду давления "масло-газ" в алгоритме АвтоНУ *)
  fb_AutoNU_Ust_Swap(StrAP:=IM.AutoNU_Ust_Swap);

  (* Уставка по перепаду давления "масло-газ" в алгоритме Тест dPmg *)
  fb_testdPmg_Ust_dPLow(StrAP:=IM.testdPmg_Ust_dPLow);

  (* Угол наклона ВНА в алгоритме Антипомпаж *)
  fb_AntiPompag_UgolVNA(StrAP:=IM.AntiPompag_UgolVNA);

  (*Коэффициент сжимаемости газа в алгоритме Антипомпаж *)
  fb_AntiPompag_K(StrAP:=IM.AntiPompag_K);

  (* Коэффициент расхода конфузора в алгоритме Антипомпаж *)
  fb_AntiPompag_A(StrAP:=IM.AntiPompag_A);

  (* Удельный вес газа в алгоритме Антипомпаж *)
  fb_AntiPompag_y0(StrAP:=IM.AntiPompag_y0);

    (* Переключатель разблокировки кранов: 1 - допстить управление кранами  *)
  fb_TypeSwitch(StrDP:=IM.TypeSwitch);

    (* Селектор выбора основной/резервный НУ  *)
  fb_AutoNU_mainNU(StrDP:=IM.AutoNU_mainNU);
END_FUNCTION_BLOCK

FUNCTION_BLOCK OPC_IM_get
  VAR_EXTERNAL
    IM : ImConfig;
    IM_SingleSignals_DverShkafaOtkryta_status : UDINT;
    IM_SingleSignals_KZ_10kv_status : UDINT;
    IM_SingleSignals_NOGPA_knopkaSHU_status : UDINT;
    IM_SingleSignals_NS_G10_G11_status : UDINT;
    IM_SingleSignals_NS_G13_G14_status : UDINT;
    IM_SingleSignals_NS_G15_G16_status : UDINT;
    IM_SingleSignals_NS_G17_status : UDINT;
    IM_SingleSignals_NS_G18_G19_status : UDINT;
    IM_SingleSignals_NS_G1_G2_status : UDINT;
    IM_SingleSignals_NS_G3_G4_status : UDINT;
    IM_SingleSignals_NS_G5_G6_status : UDINT;
    IM_SingleSignals_NS_G7_G8_status : UDINT;
    IM_SingleSignals_OsevoiSdvig_levo_status : UDINT;
    IM_SingleSignals_OsevoiSdvig_pravo_status : UDINT;
    IM_SingleSignals_P_oil_low_status : UDINT;
    IM_SingleSignals_QF10_QF11_on_status : UDINT;
    IM_SingleSignals_QF12_QF13_on_status : UDINT;
    IM_SingleSignals_QF14_QF15_on_status : UDINT;
    IM_SingleSignals_QF1_on_status : UDINT;
    IM_SingleSignals_QF22_on_status : UDINT;
    IM_SingleSignals_QF23_on_status : UDINT;
    IM_SingleSignals_QF2_on_status : UDINT;
    IM_SingleSignals_QF4_QF5_on_status : UDINT;
    IM_SingleSignals_QF6_QF7_on_status : UDINT;
    IM_SingleSignals_QF8_QF9_on_status : UDINT;
    IM_SingleSignals_Vozb_AsinchHod_status : UDINT;
    IM_SingleSignals_Vozb_ControlVozbuditela_status : UDINT;
    IM_SingleSignals_Vozb_KontaktorON_status : UDINT;
    IM_SingleSignals_Vozb_Overload_status : UDINT;
    IM_SingleSignals_Vozb_ProboiVentila_status : UDINT;
    IM_SingleSignals_Vozb_ReSynchronize_status : UDINT;
    IM_SingleSignals_dP_gazgaz_Kran1_status : UDINT;
    IM_SingleSignals_dP_oilgaz_low_status : UDINT;
    IM_Ten_inCommand_ARM : UINT;
    IM_Ten_status : UDINT;
    IM_kran1_inCommand_ARM : UINT;
    IM_kran1_status : UDINT;
    IM_kran2_inCommand_ARM : UINT;
    IM_kran2_status : UDINT;
    IM_kran3b_inCommand_ARM : UINT;
    IM_kran3b_status : UDINT;
    IM_kran4_inCommand_ARM : UINT;
    IM_kran4_status : UDINT;
    IM_kran5_inCommand_ARM : UINT;
    IM_kran5_status : UDINT;
    IM_kran6_inCommand_ARM : UINT;
    IM_kran6_status : UDINT;
    IM_mv_inCommand_ARM : UINT;
    IM_mv_status : UDINT;
    IM_nu1_inCommand_ARM : UINT;
    IM_nu1_status : UDINT;
    IM_nu2_inCommand_ARM : UINT;
    IM_nu2_status : UDINT;
    IM_pns_inCommand_ARM : UINT;
    IM_pns_status : UDINT;
    IM_v1_Avom_inCommand_ARM : UINT;
    IM_v1_Avom_status : UDINT;
    IM_v2_Avom_inCommand_ARM : UINT;
    IM_v2_Avom_status : UDINT;
    algoritms_testIm_TypeSwitch_inCommand_ARM : UINT;
    algoritms_autoNu_mainNU_inCommand_ARM : UINT;
    algoritms_AutoAvom_hysteresis_inCommand_ARM : UINT;
    algoritms_AutoAvom_hysteresis_newValue : LREAL;
    algoritms_AutoAvom_on1Temperature_inCommand_ARM : UINT;
    algoritms_AutoAvom_on1Temperature_newValue : LREAL;
    algoritms_AutoAvom_on2Temperature_inCommand_ARM : UINT;
    algoritms_AutoAvom_on2Temperature_newValue : LREAL;
    algoritms_AutoTen_offTemperature_inCommand_ARM : UINT;
    algoritms_AutoTen_offTemperature_newValue : LREAL;
    algoritms_AutoPns_Ust_Run_inCommand_ARM : UINT;
    algoritms_AutoPns_Ust_Run_newValue : LREAL;
    algoritms_AutoPns_Ust_Stop_inCommand_ARM : UINT;
    algoritms_AutoPns_Ust_Stop_newValue : LREAL;
    algoritms_puskOilSystem_Ust_dPmg_inCommand_ARM : UINT;
    algoritms_puskOilSystem_Ust_dPmg_newValue : LREAL;
    algoritms_autoNu_Ust_Swap_inCommand_ARM : UINT;
    algoritms_autoNu_Ust_Swap_newValue : LREAL;
    algoritms_AntiPompag_UgolVNA_inCommand_ARM : UINT;
    algoritms_AntiPompag_UgolVNA_newValue : LREAL;
    algoritms_testdPmg_Ust_dPLow_inCommand_ARM : UINT;
    algoritms_testdPmg_Ust_dPLow_newValue : LREAL;
    Reset_HasNU : BOOL;
    algoritms_autoNu_Reset_HasNU : BOOL;
  END_VAR

  (* OPC Get - IM. Чтение текущих состояний тэгов _______________________________________________________*)

  Im.kran1.inCommand_ARM	:= UINT_TO_WORD(IM_kran1_inCommand_ARM);
  Im.kran2.inCommand_ARM	:= UINT_TO_WORD(IM_kran2_inCommand_ARM);
  Im.kran3b.inCommand_ARM	:= UINT_TO_WORD(IM_kran3b_inCommand_ARM);
  Im.kran4.inCommand_ARM	:= UINT_TO_WORD(IM_kran4_inCommand_ARM);
  Im.kran5.inCommand_ARM	:= UINT_TO_WORD(IM_kran5_inCommand_ARM);
  Im.kran6.inCommand_ARM	:= UINT_TO_WORD(IM_kran6_inCommand_ARM);
  Im.mv.inCommand_ARM	          := UINT_TO_WORD(IM_mv_inCommand_ARM);
  Im.nu1.inCommand_ARM	:= UINT_TO_WORD(IM_nu1_inCommand_ARM);
  Im.nu2.inCommand_ARM	:= UINT_TO_WORD(IM_nu2_inCommand_ARM);
  Im.pns.inCommand_ARM	:= UINT_TO_WORD(IM_pns_inCommand_ARM);
  Im.Ten.inCommand_ARM	:= UINT_TO_WORD(IM_Ten_inCommand_ARM);
  Im.v1_Avom.inCommand_ARM	:= UINT_TO_WORD(IM_v1_Avom_inCommand_ARM);
  Im.v2_Avom.inCommand_ARM	:= UINT_TO_WORD(IM_v2_Avom_inCommand_ARM);

  Im.AutoAvom_hysteresis.newValue        := algoritms_AutoAvom_hysteresis_newValue;
  Im.AutoAvom_hysteresis.inCommand_ARM   := UINT_TO_WORD(algoritms_AutoAvom_hysteresis_inCommand_ARM);
  Im.AutoAvom_onTemp1.newValue        := algoritms_AutoAvom_on1Temperature_newValue;
  Im.AutoAvom_onTemp1.inCommand_ARM      := UINT_TO_WORD(algoritms_AutoAvom_on1Temperature_inCommand_ARM);
  Im.AutoAvom_onTemp2.newValue        := algoritms_AutoAvom_on2Temperature_newValue;
  Im.AutoAvom_onTemp2.inCommand_ARM      := UINT_TO_WORD(algoritms_AutoAvom_on2Temperature_inCommand_ARM);

  Im.AutoTen_offTemperature.newValue        := algoritms_AutoTen_offTemperature_newValue;
  Im.AutoTen_offTemperature.inCommand_ARM   := UINT_TO_WORD(algoritms_AutoTen_offTemperature_inCommand_ARM);

  Im.AutoPns_UstRun.newValue        := algoritms_AutoPns_Ust_Run_newValue;
  Im.AutoPns_UstRun.inCommand_ARM   := UINT_TO_WORD(algoritms_AutoPns_Ust_Run_inCommand_ARM);
  Im.AutoPns_UstStop.newValue        := algoritms_AutoPns_Ust_Stop_newValue;
  Im.AutoPns_UstStop.inCommand_ARM   := UINT_TO_WORD(algoritms_AutoPns_Ust_Stop_inCommand_ARM);

  Im.PuskOilSystem_UstdPmg.newValue        := algoritms_puskOilSystem_Ust_dPmg_newValue;
  Im.PuskOilSystem_UstdPmg.inCommand_ARM   := UINT_TO_WORD(algoritms_puskOilSystem_Ust_dPmg_inCommand_ARM);

  Im.AutoNU_Ust_Swap.newValue        := algoritms_autoNu_Ust_Swap_newValue;
  Im.AutoNU_Ust_Swap.inCommand_ARM   := UINT_TO_WORD(algoritms_autoNu_Ust_Swap_inCommand_ARM);

  Im.testdPmg_Ust_dPLow.newValue        := algoritms_testdPmg_Ust_dPLow_newValue;
  Im.testdPmg_Ust_dPLow.inCommand_ARM   := UINT_TO_WORD(algoritms_testdPmg_Ust_dPLow_inCommand_ARM);

  Im.AntiPompag_UgolVNA.newValue        := algoritms_AntiPompag_UgolVNA_newValue;
  Im.AntiPompag_UgolVNA.inCommand_ARM   := UINT_TO_WORD(algoritms_AntiPompag_UgolVNA_inCommand_ARM);

  Im.TypeSwitch.inCommand_ARM           := UINT_TO_WORD(algoritms_testIm_TypeSwitch_inCommand_ARM);

  Im.AutoNU_mainNU.inCommand_ARM        := UINT_TO_WORD(algoritms_autoNu_mainNU_inCommand_ARM);

  Reset_HasNU   := algoritms_autoNu_Reset_HasNU;
END_FUNCTION_BLOCK

FUNCTION_BLOCK OPC_IM_set
  VAR_EXTERNAL
    IM : ImConfig;
    IM_SingleSignals_DverShkafaOtkryta_status : UDINT;
    IM_SingleSignals_KZ_10kv_status : UDINT;
    IM_SingleSignals_NOGPA_knopkaSHU_status : UDINT;
    IM_SingleSignals_NS_G10_G11_status : UDINT;
    IM_SingleSignals_NS_G13_G14_status : UDINT;
    IM_SingleSignals_NS_G15_G16_status : UDINT;
    IM_SingleSignals_NS_G17_status : UDINT;
    IM_SingleSignals_NS_G18_G19_status : UDINT;
    IM_SingleSignals_NS_G1_G2_status : UDINT;
    IM_SingleSignals_NS_G3_G4_status : UDINT;
    IM_SingleSignals_NS_G5_G6_status : UDINT;
    IM_SingleSignals_NS_G7_G8_status : UDINT;
    IM_SingleSignals_OsevoiSdvig_levo_status : UDINT;
    IM_SingleSignals_OsevoiSdvig_pravo_status : UDINT;
    IM_SingleSignals_P_oil_low_status : UDINT;
    IM_SingleSignals_QF10_QF11_on_status : UDINT;
    IM_SingleSignals_QF12_QF13_on_status : UDINT;
    IM_SingleSignals_QF14_QF15_on_status : UDINT;
    IM_SingleSignals_QF1_on_status : UDINT;
    IM_SingleSignals_QF22_on_status : UDINT;
    IM_SingleSignals_QF23_on_status : UDINT;
    IM_SingleSignals_QF2_on_status : UDINT;
    IM_SingleSignals_QF4_QF5_on_status : UDINT;
    IM_SingleSignals_QF6_QF7_on_status : UDINT;
    IM_SingleSignals_QF8_QF9_on_status : UDINT;
    IM_SingleSignals_Vozb_AsinchHod_status : UDINT;
    IM_SingleSignals_Vozb_ControlVozbuditela_status : UDINT;
    IM_SingleSignals_Vozb_KontaktorON_status : UDINT;
    IM_SingleSignals_Vozb_Overload_status : UDINT;
    IM_SingleSignals_Vozb_ProboiVentila_status : UDINT;
    IM_SingleSignals_Vozb_ReSynchronize_status : UDINT;
    IM_SingleSignals_dP_gazgaz_Kran1_status : UDINT;
    IM_SingleSignals_dP_oilgaz_low_status : UDINT;
    IM_Ten_inCommand_ARM : UINT;
    IM_Ten_status : UDINT;
    IM_kran1_inCommand_ARM : UINT;
    IM_kran1_status : UDINT;
    IM_kran2_inCommand_ARM : UINT;
    IM_kran2_status : UDINT;
    IM_kran3b_inCommand_ARM : UINT;
    IM_kran3b_status : UDINT;
    IM_kran4_inCommand_ARM : UINT;
    IM_kran4_status : UDINT;
    IM_kran5_inCommand_ARM : UINT;
    IM_kran5_status : UDINT;
    IM_kran6_inCommand_ARM : UINT;
    IM_kran6_status : UDINT;
    IM_mv_inCommand_ARM : UINT;
    IM_mv_status : UDINT;
    IM_nu1_inCommand_ARM : UINT;
    IM_nu1_status : UDINT;
    IM_nu2_inCommand_ARM : UINT;
    IM_nu2_status : UDINT;
    IM_pns_inCommand_ARM : UINT;
    IM_pns_status : UDINT;
    IM_v1_Avom_inCommand_ARM : UINT;
    IM_v1_Avom_status : UDINT;
    IM_v2_Avom_inCommand_ARM : UINT;
    IM_v2_Avom_status : UDINT;
    algoritms_AutoAvom_hysteresis_Value : LREAL;
    algoritms_AutoAvom_hysteresis_status : UDINT;
    algoritms_AutoAvom_on1Temperature_Value : LREAL;
    algoritms_AutoAvom_on1Temperature_status : UDINT;
    algoritms_AutoAvom_on2Temperature_Value : LREAL;
    algoritms_AutoAvom_on2Temperature_status : UDINT;
    algoritms_autoNu_mainNU_status : UDINT;
    algoritms_testIm_TypeSwitch_status : UDINT;
    algoritms_AutoTen_offTemperature_Value : LREAL;
    algoritms_AutoTen_offTemperature_status : UDINT;
    algoritms_AutoPns_Ust_Run_Value : LREAL;
    algoritms_AutoPns_Ust_Run_status : UDINT;
    algoritms_AutoPns_Ust_Stop_Value : LREAL;
    algoritms_AutoPns_Ust_Stop_status : UDINT;
    algoritms_puskOilSystem_Ust_dPmg_Value : LREAL;
    algoritms_puskOilSystem_Ust_dPmg_status : UDINT;
    algoritms_autoNu_Ust_Swap_Value : LREAL;
    algoritms_autoNu_Ust_Swap_status : UDINT;
    algoritms_AntiPompag_UgolVNA_Value : LREAL;
    algoritms_AntiPompag_UgolVNA_status : UDINT;
    algoritms_testdPmg_Ust_dPLow_Value : LREAL;
    algoritms_testdPmg_Ust_dPLow_status : UDINT;
  END_VAR

  (* OPC Set - IM. Запись текущих состояний тэгов _______________________________________________________*)

  IM_kran1_status	:= DWORD_TO_UDINT(Im.kran1.status);
  IM_kran2_status	:= DWORD_TO_UDINT(Im.kran2.status);
  IM_kran3b_status	:= DWORD_TO_UDINT(Im.kran3b.status);
  IM_kran4_status	:= DWORD_TO_UDINT(Im.kran4.status);
  IM_kran5_status	:= DWORD_TO_UDINT(Im.kran5.status);
  IM_kran6_status	:= DWORD_TO_UDINT(Im.kran6.status);
  IM_mv_status	:= DWORD_TO_UDINT(Im.mv.status);
  IM_nu1_status	:= DWORD_TO_UDINT(Im.nu1.status);
  IM_nu2_status	:= DWORD_TO_UDINT(Im.nu2.status);
  IM_pns_status	:= DWORD_TO_UDINT(Im.pns.status);
  IM_Ten_status	:= DWORD_TO_UDINT(Im.Ten.status);
  IM_v1_Avom_status	:= DWORD_TO_UDINT(Im.v1_Avom.status);
  IM_v2_Avom_status	:= DWORD_TO_UDINT(Im.v2_Avom.status);
  IM_SingleSignals_NOGPA_knopkaSHU_status	:= DWORD_TO_UDINT(Im.SingleSignals.NOGPA_knopkaSHU.status);
  IM_SingleSignals_dP_gazgaz_Kran1_status	:= DWORD_TO_UDINT(Im.SingleSignals.dP_gazgaz_Kran1.status);
  IM_SingleSignals_P_oil_low_status	:= DWORD_TO_UDINT(Im.SingleSignals.P_oil_low.status);
  IM_SingleSignals_DverShkafaOtkryta_status	:= DWORD_TO_UDINT(Im.SingleSignals.DverShkafaOtkryta.status);
  IM_SingleSignals_KZ_10kv_status	:= DWORD_TO_UDINT(Im.SingleSignals.KZ_10kv.status);
  IM_SingleSignals_OsevoiSdvig_levo_status	:= DWORD_TO_UDINT(Im.SingleSignals.OsevoiSdvig_levo.status);
  IM_SingleSignals_OsevoiSdvig_pravo_status	:= DWORD_TO_UDINT(Im.SingleSignals.OsevoiSdvig_pravo.status);
  IM_SingleSignals_QF4_QF5_on_status	:= DWORD_TO_UDINT(Im.SingleSignals.QF4_QF5_on.status);
  IM_SingleSignals_QF6_QF7_on_status	:= DWORD_TO_UDINT(Im.SingleSignals.QF6_QF7_on.status);
  IM_SingleSignals_QF8_QF9_on_status	:= DWORD_TO_UDINT(Im.SingleSignals.QF8_QF9_on.status);
  IM_SingleSignals_QF10_QF11_on_status	:= DWORD_TO_UDINT(Im.SingleSignals.QF10_QF11_on.status);
  IM_SingleSignals_QF12_QF13_on_status	:= DWORD_TO_UDINT(Im.SingleSignals.QF12_QF13_on.status);
  IM_SingleSignals_QF14_QF15_on_status	:= DWORD_TO_UDINT(Im.SingleSignals.QF14_QF15_on.status);
  IM_SingleSignals_QF1_on_status	:= DWORD_TO_UDINT(Im.SingleSignals.QF1_on.status);
  IM_SingleSignals_QF2_on_status	:= DWORD_TO_UDINT(Im.SingleSignals.QF2_on.status);
  IM_SingleSignals_QF23_on_status	:= DWORD_TO_UDINT(Im.SingleSignals.QF23_on.status);
  IM_SingleSignals_Vozb_AsinchHod_status	:= DWORD_TO_UDINT(Im.SingleSignals.Vozb_AsinchHod.status);
  IM_SingleSignals_Vozb_ControlVozbuditela_status	:= DWORD_TO_UDINT(Im.SingleSignals.Vozb_ControlVozbuditela.status);
  IM_SingleSignals_Vozb_KontaktorON_status	:= DWORD_TO_UDINT(Im.SingleSignals.Vozb_KontaktorON.status);
  IM_SingleSignals_Vozb_Overload_status	:= DWORD_TO_UDINT(Im.SingleSignals.Vozb_Overload.status);
  IM_SingleSignals_Vozb_ProboiVentila_status	:= DWORD_TO_UDINT(Im.SingleSignals.Vozb_ProboiVentila.status);
  IM_SingleSignals_Vozb_ReSynchronize_status	:= DWORD_TO_UDINT(Im.SingleSignals.Vozb_ReSynchronize.status);
  IM_SingleSignals_dP_oilgaz_low_status	:= DWORD_TO_UDINT(Im.SingleSignals.dP_oilgaz_low.status);
  IM_SingleSignals_QF22_on_status	:= DWORD_TO_UDINT(Im.SingleSignals.QF22_on.status);
  IM_SingleSignals_NS_G1_G2_status	:= DWORD_TO_UDINT(Im.SingleSignals.NS_G1_G2.status);
  IM_SingleSignals_NS_G3_G4_status	:= DWORD_TO_UDINT(Im.SingleSignals.NS_G3_G4.status);
  IM_SingleSignals_NS_G5_G6_status	:= DWORD_TO_UDINT(Im.SingleSignals.NS_G5_G6.status);
  IM_SingleSignals_NS_G7_G8_status	:= DWORD_TO_UDINT(Im.SingleSignals.NS_G7_G8.status);
  IM_SingleSignals_NS_G10_G11_status	:= DWORD_TO_UDINT(Im.SingleSignals.NS_G10_G11.status);
  IM_SingleSignals_NS_G13_G14_status	:= DWORD_TO_UDINT(Im.SingleSignals.NS_G13_G14.status);
  IM_SingleSignals_NS_G15_G16_status	:= DWORD_TO_UDINT(Im.SingleSignals.NS_G15_G16.status);
  IM_SingleSignals_NS_G17_status	:= DWORD_TO_UDINT(Im.SingleSignals.NS_G17.status);
  IM_SingleSignals_NS_G18_G19_status	:= DWORD_TO_UDINT(Im.SingleSignals.NS_G18_G19.status);

  algoritms_AutoAvom_hysteresis_Value        := Im.AutoAvom_hysteresis.Value;
  algoritms_AutoAvom_hysteresis_status       := DWORD_TO_UDINT(Im.AutoAvom_hysteresis.status);
  algoritms_AutoAvom_on1Temperature_Value    := Im.AutoAvom_onTemp1.Value;
  algoritms_AutoAvom_on1Temperature_status   := DWORD_TO_UDINT(Im.AutoAvom_onTemp1.status);
  algoritms_AutoAvom_on2Temperature_Value    := Im.AutoAvom_onTemp2.Value;
  algoritms_AutoAvom_on2Temperature_status   := DWORD_TO_UDINT(Im.AutoAvom_onTemp2.status);

  algoritms_AutoTen_offTemperature_Value    := Im.AutoTen_offTemperature.Value;
  algoritms_AutoTen_offTemperature_status   := DWORD_TO_UDINT(Im.AutoTen_offTemperature.status);

  algoritms_AutoPns_Ust_Run_Value    := Im.AutoPns_UstRun.Value;
  algoritms_AutoPns_Ust_Run_status   := DWORD_TO_UDINT(Im.AutoPns_UstRun.status);
  algoritms_AutoPns_Ust_Stop_Value    := Im.AutoPns_UstStop.Value;
  algoritms_AutoPns_Ust_Stop_status   := DWORD_TO_UDINT(Im.AutoPns_UstStop.status);

  algoritms_puskOilSystem_Ust_dPmg_Value    := Im.PuskOilSystem_UstdPmg.Value;
  algoritms_puskOilSystem_Ust_dPmg_status   := DWORD_TO_UDINT(Im.PuskOilSystem_UstdPmg.status);

  algoritms_autoNu_Ust_Swap_Value    := Im.AutoNU_Ust_Swap.Value;
  algoritms_autoNu_Ust_Swap_status   := DWORD_TO_UDINT(Im.AutoNU_Ust_Swap.status);

  algoritms_testdPmg_Ust_dPLow_Value    := Im.testdPmg_Ust_dPLow.Value;
  algoritms_testdPmg_Ust_dPLow_status   := DWORD_TO_UDINT(Im.testdPmg_Ust_dPLow.status);

  algoritms_AntiPompag_UgolVNA_Value    := Im.AntiPompag_UgolVNA.Value;
  algoritms_AntiPompag_UgolVNA_status   := DWORD_TO_UDINT(Im.AntiPompag_UgolVNA.status);

  algoritms_testIm_TypeSwitch_status  :=  DWORD_TO_UDINT(Im.TypeSwitch.status);

  algoritms_autoNu_mainNU_status      :=  DWORD_TO_UDINT(Im.AutoNU_mainNU.status);
END_FUNCTION_BLOCK

FUNCTION_BLOCK fb_DiProtection_Init
  VAR_INPUT
    data_Ini : BOOL;
    delay : TIME;
    inTag : BYTE;
    inRunOnStart : BOOL;
  END_VAR
  VAR_IN_OUT
    str_DIp : struct_DiProtection;
  END_VAR
  VAR_OUTPUT
    Init : BOOL := FALSE;
  END_VAR

  (*****            Функциональный блок переинициализации структуры  AiProtection          *****)

   Init := FALSE;

      IF data_Ini THEN                            (* Параметрам требуется переинициализация. *)
          str_DIp.delay               := delay;
          str_DIp.inTag               := inTag;
          str_DIp.inRunOnStart        := inRunOnStart;

          data_Ini:=FALSE;
          Init := TRUE;
      END_IF;
      IF Init THEN
          delay:= T#0S;
          inTag:= 0;
          inRunOnStart:= FALSE;
      END_IF;
END_FUNCTION_BLOCK

FUNCTION_BLOCK fb_AiProtection_Init
  VAR_INPUT
    data_Ini : BOOL;
    controlLimit : BYTE;
    delay : TIME;
    inTag : BYTE;
    inRunOnStart : BOOL;
  END_VAR
  VAR_IN_OUT
    str_AIp : struct_AiProtection;
  END_VAR
  VAR_OUTPUT
    Init : BOOL := FALSE;
  END_VAR

  (*****            Функциональный блок переинициализации структуры  AiProtection          *****)

   Init := FALSE;

      IF data_Ini THEN                            (* Параметрам требуется переинициализация. *)
          str_AIp.controlLimit        := controlLimit;
          str_AIp.delay               := delay;
          str_AIp.inTag               := inTag;
          str_AIp.inRunOnStart        := inRunOnStart;

          data_Ini:=FALSE;
          Init := TRUE;
      END_IF;
      IF Init THEN
          controlLimit:= 0;
          delay:= T#0S;
          inTag:= 0;
          inRunOnStart:= FALSE;
      END_IF;
END_FUNCTION_BLOCK

FUNCTION_BLOCK proc_Protections_Init
  VAR_INPUT
    init : BOOL;
  END_VAR
  VAR
    stDIp_Ini : fb_DiProtection_Init;
    stAIp_Ini : fb_AiProtection_Init;
    inits : UINT;
  END_VAR
  VAR_INPUT
    initiales : UINT;
  END_VAR
  VAR_EXTERNAL
    protections : ProtectionsConfig;
  END_VAR
  VAR
    _ProtectionTags : TYPE_ProtectionTags;
    _StatusAi : TYPE_StatusAi;
  END_VAR

  inits := 0; (* Флаг необходимости инициализации структур-дескрипторов *)

  (*************************************************Стартовая инициализация DiProtection ***************************************************)
  (* Осевой сдвиг ротора вправо ≥3,7 кгс/см *)
  stDIp_Ini(data_Ini := true, delay:=T#1S, inTag:=_ProtectionTags.AOS, inRunOnStart:=TRUE, str_DIp := protections.OsevojSdvigPravyjDi);
  inits := inits + BOOL_TO_UINT(stDIp_Ini.Init);

  (* Осевой сдвиг ротора влево ≥3,7 кгс/см *)
  stDIp_Ini(data_Ini := true, delay:=T#1S, inTag:=_ProtectionTags.AOS, inRunOnStart:=TRUE, str_DIp := protections.OsevojSdvigLevyjDi);
  inits := inits + BOOL_TO_UINT(stDIp_Ini.Init);

  (* Низкий перепад давления «масло-газ» ≤1 кгс/см² *)
  stDIp_Ini(data_Ini := true, delay:=T#20S, inTag:=_ProtectionTags.AOS, inRunOnStart:=FALSE, str_DIp := protections.dP_masloGaz_LowDI);
  inits := inits + BOOL_TO_UINT(stDIp_Ini.Init);

  (* Низкое давление масла смазки ≤ 0,4 кгс/см² *)
  stDIp_Ini(data_Ini := true, delay:=T#10S, inTag:=_ProtectionTags.AOS, inRunOnStart:=FALSE, str_DIp := protections.DavlenieMaslaSmazkiDi);
  inits := inits + BOOL_TO_UINT(stDIp_Ini.Init);

  (* МВ отключен *)
  stDIp_Ini(data_Ini := true, delay:=T#1S, inTag:=_ProtectionTags.AOS, inRunOnStart:=FALSE, str_DIp := protections.mvOff);
  inits := inits + BOOL_TO_UINT(stDIp_Ini.Init);

  (* Неисправность возбудительного устройства *)
  stDIp_Ini(data_Ini := true, delay:=T#1S, inTag:=_ProtectionTags.AOS, inRunOnStart:=TRUE, str_DIp := protections.NeispravnostVozbuzhdenijaDi);
  inits := inits + BOOL_TO_UINT(stDIp_Ini.Init);

  (* Аварийный останов цеха *)
  stDIp_Ini(data_Ini := true, delay:=T#1S, inTag:=_ProtectionTags.AOS, inRunOnStart:=TRUE, str_DIp := protections.AO_KC);
  inits := inits + BOOL_TO_UINT(stDIp_Ini.Init);

  (* Аварийный останов АО ЭГПА с ПРУ *)
  stDIp_Ini(data_Ini := true, delay:=T#100MS, inTag:=_ProtectionTags.AOS, inRunOnStart:=TRUE, str_DIp := protections.AO_PRU);
  inits := inits + BOOL_TO_UINT(stDIp_Ini.Init);

  (* Аварийный останов АО ЭГПА с ШУ *)
  stDIp_Ini(data_Ini := true, delay:=T#100MS, inTag:=_ProtectionTags.AOS, inRunOnStart:=TRUE, str_DIp := protections.AO_SHU);
  inits := inits + BOOL_TO_UINT(stDIp_Ini.Init);

  (* Срабатывание БЭАО (отказ ПТС) *)
  stDIp_Ini(data_Ini := true, delay:=T#0S, inRunOnStart:=TRUE, str_DIp := protections.Srab_BEAO);
  inits := inits + BOOL_TO_UINT(stDIp_Ini.Init);

  (* Экстренный аварийный останов ЭАО ЭГПА с ПРУ *)
  stDIp_Ini(data_Ini := true, delay:=T#0S, inRunOnStart:=TRUE, str_DIp := protections.EAO_PRU);
  inits := inits + BOOL_TO_UINT(stDIp_Ini.Init);

  (* Запуск БЭАО от кнопки ЭАО ШУ *)
  stDIp_Ini(data_Ini := true, delay:=T#0S, inRunOnStart:=TRUE, str_DIp := protections.BEAO_knSHU);
  inits := inits + BOOL_TO_UINT(stDIp_Ini.Init);

  (* Сдвиг крана №1 *)
  stDIp_Ini(data_Ini := true, delay:=T#1S, inTag:=_ProtectionTags.AOS, inRunOnStart:=FALSE, str_DIp := protections.Kran1sdvig);
  inits := inits + BOOL_TO_UINT(stDIp_Ini.Init);

  (* Сдвиг крана №2 *)
  stDIp_Ini(data_Ini := true, delay:=T#1S, inTag:=_ProtectionTags.AOS, inRunOnStart:=FALSE, str_DIp := protections.Kran2sdvig);
  inits := inits + BOOL_TO_UINT(stDIp_Ini.Init);

  (*************************************************Стартовая инициализация AiProtection ***************************************************)

  (* Температура переднего опорного подшипника двигателя, т.1 *)
  stAIp_Ini(data_Ini := true, delay:=T#3S, inTag:=_ProtectionTags.AOS, inRunOnStart:=TRUE,
  controlLimit:=_StatusAi.HA, str_AIp := protections.T_perednego_opornogo_podshipnika_dvigatelia_t1_HA);
  inits := inits + BOOL_TO_UINT(stAIp_Ini.Init);

  (* Температура заднего опорного подшипника двигателя, т.2 *)
  stAIp_Ini(data_Ini := true, delay:=T#3S, inTag:=_ProtectionTags.AOS, inRunOnStart:=TRUE,
  controlLimit:=_StatusAi.HA, str_AIp := protections.T_zadnego_opornogo_podshipnika_dvigatelia_t2_HA);
  inits := inits + BOOL_TO_UINT(stAIp_Ini.Init);

  (* Температура подшипника редуктора, т1 *)
  stAIp_Ini(data_Ini := true, delay:=T#3S, inTag:=_ProtectionTags.AOS, inRunOnStart:=TRUE,
  controlLimit:=_StatusAi.HA, str_AIp := protections.T_podshipnika_reduktora_t1_HA);
  inits := inits + BOOL_TO_UINT(stAIp_Ini.Init);

  (* Температура подшипника редуктора, т2 *)
  stAIp_Ini(data_Ini := true, delay:=T#3S, inTag:=_ProtectionTags.AOS, inRunOnStart:=TRUE,
  controlLimit:=_StatusAi.HA, str_AIp := protections.T_podshipnika_reduktora_t2_HA);
  inits := inits + BOOL_TO_UINT(stAIp_Ini.Init);

  (* Температура подшипника редуктора, т3 *)
  stAIp_Ini(data_Ini := true, delay:=T#3S, inTag:=_ProtectionTags.AOS, inRunOnStart:=TRUE,
  controlLimit:=_StatusAi.HA, str_AIp := protections.T_podshipnika_reduktora_t3_HA);
  inits := inits + BOOL_TO_UINT(stAIp_Ini.Init);

  (* Температура подшипника редуктора, т4 *)
  stAIp_Ini(data_Ini := true, delay:=T#3S, inTag:=_ProtectionTags.AOS, inRunOnStart:=TRUE,
  controlLimit:=_StatusAi.HA, str_AIp := protections.T_podshipnika_reduktora_t4_HA);
  inits := inits + BOOL_TO_UINT(stAIp_Ini.Init);

  (* Температура опорного подшипника нагнетателя, т1 *)
  stAIp_Ini(data_Ini := true, delay:=T#3S, inTag:=_ProtectionTags.AOS, inRunOnStart:=TRUE,
  controlLimit:=_StatusAi.HA, str_AIp := protections.T_opornogo_podshipnika_nagnetatelia_t1_HA);
  inits := inits + BOOL_TO_UINT(stAIp_Ini.Init);

  (* Температура опорного подшипника нагнетателя, т2 *)
  stAIp_Ini(data_Ini := true, delay:=T#3S, inTag:=_ProtectionTags.AOS, inRunOnStart:=TRUE,
  controlLimit:=_StatusAi.HA, str_AIp := protections.T_opornogo_podshipnika_nagnetatelia_t2_HA);
  inits := inits + BOOL_TO_UINT(stAIp_Ini.Init);

  (* Температура опорного подшипника нагнетателя, т3 *)
  stAIp_Ini(data_Ini := true, delay:=T#3S, inTag:=_ProtectionTags.AOS, inRunOnStart:=TRUE,
  controlLimit:=_StatusAi.HA, str_AIp := protections.T_opornogo_podshipnika_nagnetatelia_t3_HA);
  inits := inits + BOOL_TO_UINT(stAIp_Ini.Init);

  (* Температура упорно опорного подшипника нагнетателя, т4 *)
  stAIp_Ini(data_Ini := true, delay:=T#3S, inTag:=_ProtectionTags.AOS, inRunOnStart:=TRUE,
  controlLimit:=_StatusAi.HA, str_AIp := protections.T_opornoupornogo_podshipnika_nagnetatelia_t4_HA);
  inits := inits + BOOL_TO_UINT(stAIp_Ini.Init);

  (* Температура газа на выходе нагнетателя *)
  stAIp_Ini(data_Ini := true, delay:=T#3S, inTag:=_ProtectionTags.AOS, inRunOnStart:=TRUE,
  controlLimit:=_StatusAi.HA, str_AIp := protections.T_gaza_na_vykhode_nagnetatelia_HA);
  inits := inits + BOOL_TO_UINT(stAIp_Ini.Init);

  (* Перепад давления "масло-газ" *)
  stAIp_Ini(data_Ini := true, delay:=T#0S, inTag:=_ProtectionTags.AOS, inRunOnStart:=FALSE,
  controlLimit:=_StatusAi.LA, str_AIp := protections.dP_maslogaz_LA);
  inits := inits + BOOL_TO_UINT(stAIp_Ini.Init);

  (* Давление масла смазки низкое *)
  stAIp_Ini(data_Ini := true, delay:=T#0S, inTag:=_ProtectionTags.AOS, inRunOnStart:=FALSE,
  controlLimit:=_StatusAi.LA, str_AIp := protections.P_masla_smazki_nizkoe_LA);
  inits := inits + BOOL_TO_UINT(stAIp_Ini.Init);

  (* Вибрация СТД т.1 *)
  stAIp_Ini(data_Ini := true, delay:=T#3S, inTag:=_ProtectionTags.AOS, inRunOnStart:=FALSE,
  controlLimit:=_StatusAi.HA, str_AIp := protections.Vibratciia_STD_t1_HA);
  inits := inits + BOOL_TO_UINT(stAIp_Ini.Init);

  (* Вибрация СТД т.2 *)
  stAIp_Ini(data_Ini := true, delay:=T#3S, inTag:=_ProtectionTags.AOS, inRunOnStart:=FALSE,
  controlLimit:=_StatusAi.HA, str_AIp := protections.Vibratciia_STD_t2_HA);
  inits := inits + BOOL_TO_UINT(stAIp_Ini.Init);

  (* Вибрация ротора нагнетателя т.1 *)
  stAIp_Ini(data_Ini := true, delay:=T#3S, inTag:=_ProtectionTags.AOS, inRunOnStart:=FALSE,
  controlLimit:=_StatusAi.HA, str_AIp := protections.Vibratciia_rotora_nagnetatelia_t1_HA);
  inits := inits + BOOL_TO_UINT(stAIp_Ini.Init);

  (* Вибрация ротора нагнетателя т.2 *)
  stAIp_Ini(data_Ini := true, delay:=T#3S, inTag:=_ProtectionTags.AOS, inRunOnStart:=FALSE,
  controlLimit:=_StatusAi.HA, str_AIp := protections.Vibratciia_rotora_nagnetatelia_t2_HA);
  inits := inits + BOOL_TO_UINT(stAIp_Ini.Init);

  (* Вибрация ротора нагнетателя т.3 *)
  stAIp_Ini(data_Ini := true, delay:=T#3S, inTag:=_ProtectionTags.AOS, inRunOnStart:=FALSE,
  controlLimit:=_StatusAi.HA, str_AIp := protections.Vibratciia_rotora_nagnetatelia_t3_HA);
  inits := inits + BOOL_TO_UINT(stAIp_Ini.Init);

  (* Вибрация ротора нагнетателя т.4 *)
  stAIp_Ini(data_Ini := true, delay:=T#3S, inTag:=_ProtectionTags.AOS, inRunOnStart:=FALSE,
  controlLimit:=_StatusAi.HA, str_AIp := protections.Vibratciia_rotora_nagnetatelia_t4_HA);
  inits := inits + BOOL_TO_UINT(stAIp_Ini.Init);

  (* Осевой сдвиг ротора нагнетателя *)
  stAIp_Ini(data_Ini := true, delay:=T#3S, inTag:=_ProtectionTags.AOS, inRunOnStart:=TRUE,
  controlLimit:=_StatusAi.HA, str_AIp := protections.Osevoi_sdvig_rotora_nagnetatelia_HA);
  inits := inits + BOOL_TO_UINT(stAIp_Ini.Init);

  (* Уровень масла в маслобаке *)
  stAIp_Ini(data_Ini := true, delay:=T#3S, inTag:=_ProtectionTags.AOS, inRunOnStart:=TRUE,
  controlLimit:=_StatusAi.LA, str_AIp := protections.Uroven_masla_v_maslobake_LA);
  inits := inits + BOOL_TO_UINT(stAIp_Ini.Init);

  IF init THEN initiales := inits; END_IF;
END_FUNCTION_BLOCK

FUNCTION_BLOCK fb_DiProtection
  VAR_INPUT
    di : struct_singleSignal;
  END_VAR
  VAR_IN_OUT
    StrDIp : struct_DiProtection;
  END_VAR
  VAR
    _sunpackerCommand : fb_sunpackerCommand;
    _ProtectionTags : TYPE_ProtectionTags;
    _signalingTp : TOF;
    timer : TON;
    SignalingTrig : R_TRIG;
    SignalingFTrig : F_TRIG;
    SignalingDi : BOOL;
    source : BYTE;
    cmd : BYTE;
    lastCmd : BYTE;
    source_for_Status : BYTE;
    cmd_for_Status : BYTE;
    command_error_for_Status : BYTE;
    resetCmdTimer : TON;
    resetCmdTimerPriznak : BOOL;
    signalinTimer : TON;
    runOnStart_Trig : R_TRIG;
  END_VAR

  timer(IN := di.Q AND StrDIp.isRunning  , PT := StrDIp.delay);
  SignalingTrig(CLK := timer.Q);
  IF SignalingTrig.Q THEN
  	SignalingDi := TRUE;
  END_IF;
  SignalingFTrig(CLK := timer.Q);
  IF SignalingFTrig.Q THEN
  	SignalingDi := FALSE;
  END_IF;

  StrDIp.Tag := StrDIp.inTag;
  StrDIp.RunOnStart := StrDIp.inRunOnStart;

  StrDIp.CanRun := StrDIp.inCanRun;

  StrDIp.OpcCommandsDisabled := StrDIp.inOpcCommandsDisabled;

  (* ---- Если управление с ВУ заблокировано, то передаем команду из алгоритма ---- *)
  IF StrDIp.inOpcCommandsDisabled THEN
  	StrDIp.inCommand := StrDIp.inCommand_Alg;
  ELSE (* иначе передаем команду с АРМа*)
  	StrDIp.inCommand := StrDIp.inCommand_ARM;
  END_IF;

  _sunpackerCommand(command := StrDIp.inCommand);
  	source := _sunpackerCommand.source;
  	cmd := _sunpackerCommand.cmd;

  IF cmd <> 0 AND lastCmd <> cmd AND (((NOT StrDIp.opcCommandsDisabled) AND source > 0) OR source = 0) then

  	CASE BYTE_TO_INT(cmd) OF
  	        (*cmdRun*) 1: 	IF        NOT StrDIp.Remont THEN
  					StrDIp.isEnded := FALSE;
  					StrDIp.hasError 	:= FALSE;
  					StrDIp.isRunning := TRUE;
  					cmd_for_Status := cmd;
  					source_for_Status := source;
  					command_error_for_Status := 0;
  				ELSE
  					StrDIp.isRunning := FALSE;
  					StrDIp.isEnded := FALSE;
  					StrDIp.hasError 	:= FALSE;

  					cmd_for_Status := 0;
  					source_for_Status := source;
  					command_error_for_Status := cmd;
  				END_IF;
                                          StrDIp.inOpcCommandsDisabled:=FALSE;

                  (*cmdReset*) 2: 	StrDIp.isRunning := FALSE;
  				StrDIp.isEnded := FALSE;
  				StrDIp.hasError 	:= FALSE;
  				SignalingDi:= FALSE;
  				StrDIp.Check := FALSE;
  				cmd_for_Status := cmd;
  				source_for_Status := source;
  				command_error_for_Status := 0;
                                         StrDIp.inOpcCommandsDisabled:=FALSE;

  	(*cmd_setRemont*) 4 :	StrDIp.Remont := TRUE;
  				(*StrDIp.isRunning := FALSE;*)

  				cmd_for_Status := cmd;
  				source_for_Status := source;
  				command_error_for_Status := 0;
          (*cmd_resetRemont*) 5 : 	(*IF di.Q THEN
  					cmd_for_Status := 0;
  					source_for_Status := 0;
  					command_error_for_Status := cmd;
  				ELSE*)
  					StrDIp.Remont := FALSE;
  					(*StrDIp.isRunning := TRUE;*)

  					cmd_for_Status := cmd;
  					source_for_Status := source;
  					command_error_for_Status := 0;
  				(*END_IF;*)
  	(*cmd_setCheck*) 6 : 	StrDIp.Check := TRUE;

  				cmd_for_Status := cmd;
  				source_for_Status := source;
  				command_error_for_Status := 0;
  	END_CASE;
  	resetCmdTimer(IN := false);
  	resetCmdTimerPriznak := TRUE;
  END_IF;
  lastCmd := cmd;

  resetCmdTimer(IN := resetCmdTimerPriznak);
  IF resetCmdTimer.Q THEN
  	resetCmdTimerPriznak := FALSE;
  	source_for_Status := 0;
  	cmd_for_Status := 0;
  	command_error_for_Status := 0;
  END_IF;

  IF StrDIp.isRunning AND NOT StrDIp.Remont AND NOT StrDIp.Check THEN
  	StrDIp.Signaling := SignalingDi;
  	StrDIp.SignalingTP := _signalingTp.Q;
  ELSE
  	StrDIp.Signaling := 0;
  	StrDIp.SignalingTP := 0;
  END_IF;

  _signalingTp(in := StrDIp.Signaling, PT := T#1s);

  StrDIp.status :=  SHL(BYTE_TO_DWORD(source_for_Status), 29)
  			OR SHL(BYTE_TO_DWORD(cmd_for_Status), 26)
  			OR SHL(BYTE_TO_DWORD(command_error_for_Status), 23)
  			OR SHL(BOOL_TO_DWORD(StrDIp.OpcCommandsDisabled ), 21)
  			OR SHL(BOOL_TO_DWORD(StrDIp.Signaling), 16)
  			OR SHL(BOOL_TO_DWORD(StrDIp.RunOnStart ), 15)
  			OR SHL(BOOL_TO_DWORD(StrDIp.remont), 6)
  			OR SHL(BOOL_TO_DWORD(StrDIp.Check), 5)
  			OR SHL(BOOL_TO_DWORD(StrDIp.hasError), 4)
  			OR SHL(BOOL_TO_DWORD(StrDIp.SignalingTP), 3)
  			OR SHL(BOOL_TO_DWORD(StrDIp.CanRun), 2)
  			OR SHL(BOOL_TO_DWORD(StrDIp.isEnded), 1)
  			OR BOOL_TO_DWORD(StrDIp.isRunning);
END_FUNCTION_BLOCK

FUNCTION_BLOCK fb_MvProtection
  VAR_INPUT
    sw : struct_SectionSwitch;
  END_VAR
  VAR_IN_OUT
    StrDIp : struct_DiProtection;
  END_VAR
  VAR
    _sunpackerCommand : fb_sunpackerCommand;
    statusDualInput : TYPE_statusDualInput;
    _ProtectionTags : TYPE_ProtectionTags;
    _signalingTp : TOF;
    timer : TON;
    SignalingTrig : R_TRIG;
    SignalingFTrig : F_TRIG;
    SignalingDi : BOOL;
    source : BYTE;
    cmd : BYTE;
    lastCmd : BYTE;
    source_for_Status : BYTE;
    cmd_for_Status : BYTE;
    command_error_for_Status : BYTE;
    resetCmdTimer : TON;
    resetCmdTimerPriznak : BOOL;
    signalinTimer : TON;
    runOnStart_Trig : R_TRIG;
  END_VAR

  timer(IN := (sw.onStatus = statusDualInput.STATUS_OFF) AND StrDIp.isRunning  , PT := StrDIp.delay);
  SignalingTrig(CLK := timer.Q);
  IF SignalingTrig.Q THEN
  	SignalingDi := TRUE;
  END_IF;
  SignalingFTrig(CLK := timer.Q);
  IF SignalingFTrig.Q THEN
  	SignalingDi := FALSE;
  END_IF;

  StrDIp.Tag := StrDIp.inTag;
  StrDIp.RunOnStart := StrDIp.inRunOnStart;

  StrDIp.CanRun := StrDIp.inCanRun;

  StrDIp.OpcCommandsDisabled := StrDIp.inOpcCommandsDisabled;

  (* ---- Если управление с ВУ заблокировано, то передаем команду из алгоритма ---- *)
  IF StrDIp.inOpcCommandsDisabled THEN
  	StrDIp.inCommand := StrDIp.inCommand_Alg;
  ELSE (* иначе передаем команду с АРМа*)
  	StrDIp.inCommand := StrDIp.inCommand_ARM;
  END_IF;

  _sunpackerCommand(command := StrDIp.inCommand);
  	source := _sunpackerCommand.source;
  	cmd := _sunpackerCommand.cmd;

  IF cmd <> 0 AND lastCmd <> cmd AND (((NOT StrDIp.opcCommandsDisabled) AND source > 0) OR source = 0) then
  	CASE BYTE_TO_INT(cmd) OF
  	        (*cmdRun*) 1: 	IF        NOT StrDIp.Remont THEN
  					StrDIp.isEnded := FALSE;
  					StrDIp.hasError 	:= FALSE;
  					StrDIp.isRunning := TRUE;
  					cmd_for_Status := cmd;
  					source_for_Status := source;
  					command_error_for_Status := 0;
  				ELSE
  					StrDIp.isRunning := FALSE;
  					StrDIp.isEnded := FALSE;
  					StrDIp.hasError 	:= FALSE;

  					cmd_for_Status := 0;
  					source_for_Status := source;
  					command_error_for_Status := cmd;
  				END_IF;
                                          StrDIp.inOpcCommandsDisabled:=FALSE;

                  (*cmdReset*) 2: 	StrDIp.isRunning := FALSE;
  				StrDIp.isEnded := FALSE;
  				StrDIp.hasError 	:= FALSE;
  				SignalingDi:= FALSE;
  				StrDIp.Check := FALSE;
  				cmd_for_Status := cmd;
  				source_for_Status := source;
  				command_error_for_Status := 0;
                                          StrDIp.inOpcCommandsDisabled:=FALSE;

  	(*cmd_setRemont*) 4 :	StrDIp.Remont := TRUE;
  				(*StrDIp.isRunning := FALSE;*)

  				cmd_for_Status := cmd;
  				source_for_Status := source;
  				command_error_for_Status := 0;

          (*cmd_resetRemont*) 5 : 	(*IF (sw.onStatus = statusDualInput.STATUS_OFF) THEN
  					cmd_for_Status := 0;
  					source_for_Status := 0;
  					command_error_for_Status := cmd;
  				ELSE*)
  					StrDIp.Remont := FALSE;
  					(*StrDIp.isRunning := TRUE;*)

  					cmd_for_Status := cmd;
  					source_for_Status := source;
  					command_error_for_Status := 0;
  				(*END_IF;*)

  	(*cmd_setCheck*) 6 : 	StrDIp.Check := TRUE;

  				cmd_for_Status := cmd;
  				source_for_Status := source;
  				command_error_for_Status := 0;
  	END_CASE;
  	resetCmdTimer(IN := false);
  	resetCmdTimerPriznak := TRUE;
  END_IF;
  lastCmd := cmd;

  resetCmdTimer(IN := resetCmdTimerPriznak);
  IF resetCmdTimer.Q THEN
  	resetCmdTimerPriznak := FALSE;
  	source_for_Status := 0;
  	cmd_for_Status := 0;
  	command_error_for_Status := 0;
  END_IF;

  IF StrDIp.isRunning AND  NOT StrDIp.Remont AND NOT StrDIp.Check THEN
  	StrDIp.Signaling := SignalingDi;
  	StrDIp.SignalingTP := _signalingTp.Q;
  ELSE
  	StrDIp.Signaling := 0;
  	StrDIp.SignalingTP := 0;
  END_IF;

  _signalingTp(in := StrDIp.Signaling, PT := T#1s);

  StrDIp.status :=  SHL(BYTE_TO_DWORD(source_for_Status), 29)
  			OR SHL(BYTE_TO_DWORD(cmd_for_Status), 26)
  			OR SHL(BYTE_TO_DWORD(command_error_for_Status), 23)
  			OR SHL(BOOL_TO_DWORD(StrDIp.OpcCommandsDisabled ), 21)
  			OR SHL(BOOL_TO_DWORD(StrDIp.Signaling), 16)
  			OR SHL(BOOL_TO_DWORD(StrDIp.RunOnStart ), 15)
  			OR SHL(BOOL_TO_DWORD(StrDIp.remont), 6)
  			OR SHL(BOOL_TO_DWORD(StrDIp.Check), 5)
  			OR SHL(BOOL_TO_DWORD(StrDIp.hasError), 4)
  			OR SHL(BOOL_TO_DWORD(StrDIp.SignalingTP), 3)
  			OR SHL(BOOL_TO_DWORD(StrDIp.CanRun), 2)
  			OR SHL(BOOL_TO_DWORD(StrDIp.isEnded), 1)
  			OR BOOL_TO_DWORD(StrDIp.isRunning);
END_FUNCTION_BLOCK

FUNCTION_BLOCK fb_KranOpenProtection
  VAR_INPUT
    im : struct_Kran;
  END_VAR
  VAR_IN_OUT
    StrDIp : struct_DiProtection;
  END_VAR
  VAR
    _sunpackerCommand : fb_sunpackerCommand;
    statusDualInput : TYPE_statusDualInput;
    _ProtectionTags : TYPE_ProtectionTags;
    _signalingTp : TOF;
    timer : TON;
    SignalingTrig : R_TRIG;
    SignalingFTrig : F_TRIG;
    SignalingDi : BOOL;
    source : BYTE;
    cmd : BYTE;
    lastCmd : BYTE;
    source_for_Status : BYTE;
    cmd_for_Status : BYTE;
    command_error_for_Status : BYTE;
    resetCmdTimer : TON;
    resetCmdTimerPriznak : BOOL;
    signalinTimer : TON;
    runOnStart_Trig : R_TRIG;
  END_VAR

  timer(IN := (im.onStatus<>statusDualInput.STATUS_ON) AND StrDIp.isRunning  , PT := StrDIp.delay);
  SignalingTrig(CLK := timer.Q);
  IF SignalingTrig.Q THEN
  	SignalingDi := TRUE;
  END_IF;
  SignalingFTrig(CLK := timer.Q);
  IF SignalingFTrig.Q THEN
  	SignalingDi := FALSE;
  END_IF;

  StrDIp.Tag := StrDIp.inTag;
  StrDIp.RunOnStart := StrDIp.inRunOnStart;

  StrDIp.CanRun := StrDIp.inCanRun;

  StrDIp.OpcCommandsDisabled := StrDIp.inOpcCommandsDisabled;

  (* ---- Если управление с ВУ заблокировано, то передаем команду из алгоритма ---- *)
  IF StrDIp.inOpcCommandsDisabled THEN
  	StrDIp.inCommand := StrDIp.inCommand_Alg;
  ELSE (* иначе передаем команду с АРМа*)
  	StrDIp.inCommand := StrDIp.inCommand_ARM;
  END_IF;

  _sunpackerCommand(command := StrDIp.inCommand);
  	source := _sunpackerCommand.source;
  	cmd := _sunpackerCommand.cmd;

  IF cmd <> 0 AND lastCmd <> cmd AND (((NOT StrDIp.opcCommandsDisabled) AND source > 0) OR source = 0) then
  	CASE BYTE_TO_INT(cmd) OF
  	        (*cmdRun*) 1: 	IF        NOT StrDIp.Remont THEN
  					StrDIp.isEnded := FALSE;
  					StrDIp.hasError 	:= FALSE;
  					StrDIp.isRunning := TRUE;
  					cmd_for_Status := cmd;
  					source_for_Status := source;
  					command_error_for_Status := 0;
  				ELSE
  					StrDIp.isRunning := FALSE;
  					StrDIp.isEnded := FALSE;
  					StrDIp.hasError 	:= FALSE;

  					cmd_for_Status := 0;
  					source_for_Status := source;
  					command_error_for_Status := cmd;
  				END_IF;
                                          StrDIp.inOpcCommandsDisabled:=FALSE;

                  (*cmdReset*) 2: 	StrDIp.isRunning := FALSE;
  				StrDIp.isEnded := FALSE;
  				StrDIp.hasError 	:= FALSE;
  				SignalingDi:= FALSE;
  				StrDIp.Check := FALSE;
  				cmd_for_Status := cmd;
  				source_for_Status := source;
  				command_error_for_Status := 0;
                                          StrDIp.inOpcCommandsDisabled:=FALSE;

  	(*cmd_setRemont*) 4 :	StrDIp.Remont := TRUE;
  				(*StrDIp.isRunning := FALSE;*)

  				cmd_for_Status := cmd;
  				source_for_Status := source;
  				command_error_for_Status := 0;

          (*cmd_resetRemont*) 5 : 	(*IF (im.onStatus<>statusDualInput.STATUS_ON) THEN
  					cmd_for_Status := 0;
  					source_for_Status := 0;
  					command_error_for_Status := cmd;
  				ELSE*)
  					StrDIp.Remont := FALSE;
  					(*StrDIp.isRunning := TRUE;*)

  					cmd_for_Status := cmd;
  					source_for_Status := source;
  					command_error_for_Status := 0;
  				(*END_IF;*)

  	(*cmd_setCheck*) 6 : 	StrDIp.Check := TRUE;

  				cmd_for_Status := cmd;
  				source_for_Status := source;
  				command_error_for_Status := 0;
  	END_CASE;
  	resetCmdTimer(IN := false);
  	resetCmdTimerPriznak := TRUE;
  END_IF;
  lastCmd := cmd;

  resetCmdTimer(IN := resetCmdTimerPriznak);
  IF resetCmdTimer.Q THEN
  	resetCmdTimerPriznak := FALSE;
  	source_for_Status := 0;
  	cmd_for_Status := 0;
  	command_error_for_Status := 0;
  END_IF;

  IF StrDIp.isRunning AND  NOT StrDIp.Remont AND NOT StrDIp.Check THEN
  	StrDIp.Signaling := SignalingDi;
  	StrDIp.SignalingTP := _signalingTp.Q;
  ELSE
  	StrDIp.Signaling := 0;
  	StrDIp.SignalingTP := 0;
  END_IF;

  _signalingTp(in := StrDIp.Signaling, PT := T#1s);

  StrDIp.status :=  SHL(BYTE_TO_DWORD(source_for_Status), 29)
  			OR SHL(BYTE_TO_DWORD(cmd_for_Status), 26)
  			OR SHL(BYTE_TO_DWORD(command_error_for_Status), 23)
  			OR SHL(BOOL_TO_DWORD(StrDIp.OpcCommandsDisabled ), 21)
  			OR SHL(BOOL_TO_DWORD(StrDIp.Signaling), 16)
  			OR SHL(BOOL_TO_DWORD(StrDIp.RunOnStart ), 15)
  			OR SHL(BOOL_TO_DWORD(StrDIp.remont), 6)
  			OR SHL(BOOL_TO_DWORD(StrDIp.Check), 5)
  			OR SHL(BOOL_TO_DWORD(StrDIp.hasError), 4)
  			OR SHL(BOOL_TO_DWORD(StrDIp.SignalingTP), 3)
  			OR SHL(BOOL_TO_DWORD(StrDIp.CanRun), 2)
  			OR SHL(BOOL_TO_DWORD(StrDIp.isEnded), 1)
  			OR BOOL_TO_DWORD(StrDIp.isRunning);
END_FUNCTION_BLOCK

FUNCTION_BLOCK fb_AiProtection
  VAR_INPUT
    ai : struct_AI;
  END_VAR
  VAR_IN_OUT
    StrAIp : struct_AiProtection;
  END_VAR
  VAR
    _sunpackerCommand : fb_sunpackerCommand;
    _signalingTp : TOF;
    _statusAi : TYPE_StatusAi;
    source : BYTE;
    cmd : BYTE;
    lastCmd : BYTE;
    source_for_Status : BYTE;
    cmd_for_Status : BYTE;
    command_error_for_Status : BYTE;
    resetCmdTimer : TON;
    resetCmdTimerPriznak : BOOL;
    signalinTimer : TON;
    timer : TON;
    SignalingTrig : R_TRIG;
    SignalingFTrig : F_TRIG;
    SignalingAi : BOOL;
  END_VAR

  timer(IN :=(ai.interval=StrAIp.controlLimit) AND (ai.interval >= _statusAi.normal) AND StrAIp.isRunning, PT :=StrAIp.delay);
  SignalingTrig(CLK := timer.Q);
  IF SignalingTrig.Q THEN
  	SignalingAi := TRUE;
  END_IF;
  SignalingFTrig(CLK := timer.Q);
  IF SignalingFTrig.Q THEN
  	SignalingAi := FALSE;
  END_IF;

  StrAIp.Tag := StrAIp.inTag;
  StrAIp.RunOnStart := StrAIp.inRunOnStart;

  StrAIp.CanRun := StrAIp.inCanRun;

  StrAIp.OpcCommandsDisabled := StrAIp.inOpcCommandsDisabled;

  (* ---- Если управление с ВУ заблокировано, то передаем команду из алгоритма ---- *)
  IF StrAIp.inOpcCommandsDisabled THEN
  	StrAIp.inCommand := StrAIp.inCommand_Alg;
  ELSE (* иначе передаем команду с АРМа*)
  	StrAIp.inCommand := StrAIp.inCommand_ARM;
  END_IF;

  _sunpackerCommand(command := StrAIp.inCommand);
  	source := _sunpackerCommand.source;
  	cmd := _sunpackerCommand.cmd;

  IF cmd <> 0 AND lastCmd <> cmd AND (((NOT StrAIp.opcCommandsDisabled) AND source > 0) OR source = 0) then

  	CASE BYTE_TO_INT(cmd) OF
  		(*cmdRun*) 1: 	IF        NOT StrAIp.Remont THEN
  					StrAIp.isEnded := FALSE;
  					StrAIp.hasError 	:= FALSE;
  					StrAIp.isRunning := TRUE;

  					cmd_for_Status := cmd;
  					source_for_Status := source;
  					command_error_for_Status := 0;
  				ELSE
  					StrAIp.isRunning := FALSE;
  					StrAIp.isEnded := FALSE;
  					StrAIp.hasError 	:= FALSE;

  					cmd_for_Status := 0;
  					source_for_Status := source;
  					command_error_for_Status := cmd;
  				END_IF;
                                          StrAIp.inopcCommandsDisabled:=FALSE;

  		(*cmdReset*) 2: 	StrAIp.isRunning := FALSE;
  				StrAIp.isEnded := FALSE;
  				StrAIp.hasError 	:= FALSE;
  				SignalingAi := FALSE;
  				StrAIp.Check := FALSE;
                                          (*StrAIp.Remont := FALSE;*)
  				cmd_for_Status := cmd;
  				source_for_Status := source;
  				command_error_for_Status := 0;
                                          StrAIp.inopcCommandsDisabled:=FALSE;

  	(*cmd_setRemont*) 4 :	StrAIp.Remont := TRUE;
  				(*StrAIp.isRunning := FALSE;*)

  				cmd_for_Status := cmd;
  				source_for_Status := source;
  				command_error_for_Status := 0;
  	(*cmd_resetRemont*) 5 : 	(*IF (ai.interval=StrAIp.controlLimit) THEN
  					cmd_for_Status := 0;
  					source_for_Status := 0;
  					command_error_for_Status := cmd;
  				ELSE*)
  					StrAIp.Remont := FALSE;
  					(*StrAIp.isRunning := TRUE;*)

  					cmd_for_Status := cmd;
  					source_for_Status := source;
  					command_error_for_Status := 0;
  				(*END_IF;*)
  	(*cmd_setCheck*) 6 : 	StrAIp.Check := TRUE;

  				cmd_for_Status := cmd;
  				source_for_Status := source;
  				command_error_for_Status := 0;
  	END_CASE;
  	resetCmdTimer(IN := false);
  	resetCmdTimerPriznak := TRUE;
  END_IF;
  lastCmd := cmd;

  resetCmdTimer(IN := resetCmdTimerPriznak);
  IF resetCmdTimer.Q THEN
  	resetCmdTimerPriznak := FALSE;
  	source_for_Status := 0;
  	cmd_for_Status := 0;
  	command_error_for_Status := 0;
  END_IF;

  IF StrAIp.isRunning AND NOT StrAIp.Remont AND NOT StrAIp.Check THEN
  	StrAIp.Signaling := SignalingAi;
  	StrAIp.SignalingTP := _signalingTp.Q;
  ELSE
  	StrAIp.Signaling := 0;
  	StrAIp.SignalingTP := 0;
  END_IF;

  _signalingTp(in := StrAIp.Signaling, PT := T#1s);

  StrAIp.status :=  SHL(BYTE_TO_DWORD(source_for_Status), 29)
  			OR SHL(BYTE_TO_DWORD(cmd_for_Status), 26)
  			OR SHL(BYTE_TO_DWORD(command_error_for_Status), 23)
  			OR SHL(BOOL_TO_DWORD(StrAIp.OpcCommandsDisabled ), 21)
  			OR SHL(BOOL_TO_DWORD(StrAIp.Signaling), 16)
  			OR SHL(BOOL_TO_DWORD(StrAIp.RunOnStart ), 15)
  			OR SHL(BOOL_TO_DWORD(StrAIp.remont), 6)
  			OR SHL(BOOL_TO_DWORD(StrAIp.Check), 5)
  			OR SHL(BOOL_TO_DWORD(StrAIp.hasError), 4)
  			OR SHL(BOOL_TO_DWORD(StrAIp.SignalingTP), 3)
  			OR SHL(BOOL_TO_DWORD(StrAIp.CanRun), 2)
  			OR SHL(BOOL_TO_DWORD(StrAIp.isEnded), 1)
  			OR BOOL_TO_DWORD(StrAIp.isRunning);
END_FUNCTION_BLOCK

FUNCTION_BLOCK proc_Protection
  VAR
    fb_OsevojSdvigPravyjDi : fb_DiProtection;
    fb_OsevojSdvigLevyjDi : fb_DiProtection;
    fb_dP_masloGaz_LowDI : fb_DiProtection;
    fb_DavlenieMaslaSmazkiDi : fb_DiProtection;
    fb_mvOff : fb_MvProtection;
    fb_NeispravnostVozbuzhdenijaDi : fb_DiProtection;
    fb_AO_KcDi : fb_DiProtection;
    fb_AO_PRU : fb_DiProtection;
    fb_AO_SHU : fb_DiProtection;
    fb_Srab_BEAO : fb_DiProtection;
    fb_EAO_PRU : fb_DiProtection;
    fb_BEAO_knSHU : fb_DiProtection;
    fb_Kran1sdvig : fb_KranOpenProtection;
    fb_Kran2sdvig : fb_KranOpenProtection;
    fb_T_per_opor_pod_dvigatelia_t1_HA : fb_AiProtection;
    fb_T_zad_opor_pod_dvigatelia_t2_HA : fb_AiProtection;
    fb_T_podshipnika_reduktora_t1_HA : fb_AiProtection;
    fb_T_podshipnika_reduktora_t2_HA : fb_AiProtection;
    fb_T_podshipnika_reduktora_t3_HA : fb_AiProtection;
    fb_T_podshipnika_reduktora_t4_HA : fb_AiProtection;
    fb_T_opor_pod_nagnetatelia_t1_HA : fb_AiProtection;
    fb_T_opor_pod_nagnetatelia_t2_HA : fb_AiProtection;
    fb_T_opor_pod_nagnetatelia_t3_HA : fb_AiProtection;
    fb_T_opor_pod_nagnetatelia_t4_HA : fb_AiProtection;
    fb_T_gaza_na_vykhode_nagnetatelia_HA : fb_AiProtection;
    fb_dP_maslogaz_LA : fb_AiProtection;
    fb_P_masla_smazki_nizkoe_LA : fb_AiProtection;
    fb_Vibratciia_STD_t1_HA : fb_AiProtection;
    fb_Vibratciia_STD_t2_HA : fb_AiProtection;
    fb_Vibratciia_rotora_nagnetatelia_t1_HA : fb_AiProtection;
    fb_Vibratciia_rotora_nagnetatelia_t2_HA : fb_AiProtection;
    fb_Vibratciia_rotora_nagnetatelia_t3_HA : fb_AiProtection;
    fb_Vibratciia_rotora_nagnetatelia_t4_HA : fb_AiProtection;
    fb_Osevoi_sdvig_rotora_nagnetatelia_HA : fb_AiProtection;
    fb_Uroven_masla_v_maslobake_LA : fb_AiProtection;
  END_VAR
  VAR_EXTERNAL
    protections : ProtectionsConfig;
    ai : AiConfig;
    IM : ImConfig;
  END_VAR

  (************************************************************* DiProtection ************************************************************)
  (* Осевой сдвиг ротора вправо ≥3,7 кгс/см *)
  fb_OsevojSdvigPravyjDi(di := IM.SingleSignals.OsevoiSdvig_pravo, StrDIp := protections.OsevojSdvigPravyjDi);

  (* Осевой сдвиг ротора влево ≥3,7 кгс/см *)
  fb_OsevojSdvigLevyjDi(di := IM.SingleSignals.OsevoiSdvig_levo, StrDIp := protections.OsevojSdvigLevyjDi);

  (* Низкий перепад давления «масло-газ» ≤1 кгс/см² *)
  fb_dP_masloGaz_LowDI(di := IM.SingleSignals.dP_oilgaz_low, StrDIp := protections.dP_masloGaz_LowDI);

  (* Низкое давление масла смазки ≤ 0,4 кгс/см² *)
  fb_DavlenieMaslaSmazkiDi(di := IM.SingleSignals.P_oil_low, StrDIp := protections.DavlenieMaslaSmazkiDi);

  (* МВ отключен *)
  fb_mvOff(sw:=IM.mv, StrDIp := protections.mvOff);

  (* Неисправность возбудительного устройства *)
  fb_NeispravnostVozbuzhdenijaDi(di := IM.SingleSignals.NS_Vozbyditela, StrDIp := protections.NeispravnostVozbuzhdenijaDi);

  (* Аварийный останов цеха *)
  fb_AO_KcDi(di := IM.SingleSignals.AO_KC, StrDIp := protections.AO_KC);

  (* Аварийный останов АО ЭГПА с ПРУ *)
  fb_AO_PRU(di := IM.SingleSignals.AOGPA_PRU, StrDIp := protections.AO_PRU);

  (* Аварийный останов АО ЭГПА с ШУ *)
  fb_AO_SHU(di := IM.SingleSignals.AOGPA_knopkaSHU, StrDIp := protections.AO_SHU);

  (* Срабатывание БЭАО (отказ ПТС) *)
  fb_Srab_BEAO(di := IM.SingleSignals.BEO_Srabat, StrDIp := protections.Srab_BEAO);

  (* Экстренный аварийный останов ЭАО ЭГПА с ПРУ *)
  fb_EAO_PRU(di := IM.SingleSignals.BEO_ON_knopkaPRU, StrDIp := protections.EAO_PRU);

  (* Запуск БЭАО от кнопки ЭАО ШУ *)
  fb_BEAO_knSHU(di := IM.SingleSignals.BEO_ON_knopkaSHU, StrDIp := protections.BEAO_knSHU);

  (* Сдвиг крана №1 *)
  fb_Kran1sdvig(im:=IM.Kran1, StrDIp := protections.Kran1sdvig);

  (* Сдвиг крана №2 *)
  fb_Kran2sdvig(im:=IM.Kran2, StrDIp := protections.Kran2sdvig);

  (************************************************************* AiProtection ************************************************************)

  (* Температура переднего опорного подшипника двигателя, т.1 *)
  fb_T_per_opor_pod_dvigatelia_t1_HA(ai := ai.T_perednego_opornogo_podshipnika_dvigatelia_t1, StrAIp := protections.T_perednego_opornogo_podshipnika_dvigatelia_t1_HA);

  (* Температура заднего опорного подшипника двигателя, т.2 *)
  fb_T_zad_opor_pod_dvigatelia_t2_HA(ai := ai.T_zadnego_opornogo_podshipnika_dvigatelia_t2, StrAIp := protections.T_zadnego_opornogo_podshipnika_dvigatelia_t2_HA);

  (* Температура подшипника редуктора, т1 *)
  fb_T_podshipnika_reduktora_t1_HA(ai := ai.T_podshipnika_reduktora_t1, StrAIp := protections.T_podshipnika_reduktora_t1_HA);

  (* Температура подшипника редуктора, т2 *)
  fb_T_podshipnika_reduktora_t2_HA(ai := ai.T_podshipnika_reduktora_t2, StrAIp := protections.T_podshipnika_reduktora_t2_HA);

  (* Температура подшипника редуктора, т3 *)
  fb_T_podshipnika_reduktora_t3_HA(ai := ai.T_podshipnika_reduktora_t3, StrAIp := protections.T_podshipnika_reduktora_t3_HA);

  (* Температура подшипника редуктора, т4 *)
  fb_T_podshipnika_reduktora_t4_HA(ai := ai.T_podshipnika_reduktora_t4, StrAIp := protections.T_podshipnika_reduktora_t4_HA);

  (* Температура опорного подшипника нагнетателя, т1 *)
  fb_T_opor_pod_nagnetatelia_t1_HA(ai := ai.T_opornogo_podshipnika_nagnetatelia_t1, StrAIp := protections.T_opornogo_podshipnika_nagnetatelia_t1_HA);

  (* Температура опорного подшипника нагнетателя, т2 *)
  fb_T_opor_pod_nagnetatelia_t2_HA(ai := ai.T_opornogo_podshipnika_nagnetatelia_t2, StrAIp := protections.T_opornogo_podshipnika_nagnetatelia_t2_HA);

  (* Температура опорного подшипника нагнетателя, т3 *)
  fb_T_opor_pod_nagnetatelia_t3_HA(ai := ai.T_opornogo_podshipnika_nagnetatelia_t3, StrAIp := protections.T_opornogo_podshipnika_nagnetatelia_t3_HA);

  (* Температура упорно опорного подшипника нагнетателя, т4 *)
  fb_T_opor_pod_nagnetatelia_t4_HA(ai := ai.T_oporno_upornogo_podshipnika_nagnetatelia_t4, StrAIp := protections.T_opornoupornogo_podshipnika_nagnetatelia_t4_HA);

  (* Температура газа на выходе нагнетателя *)
  fb_T_gaza_na_vykhode_nagnetatelia_HA(ai := ai.T_gaz_out_nagnetatelia, StrAIp := protections.T_gaza_na_vykhode_nagnetatelia_HA);

  (* Перепад давления "масло-газ" *)
  fb_dP_maslogaz_LA(ai := ai.dPmaslo_gaz, StrAIp := protections.dP_maslogaz_LA);

  (* Давление масла смазки низкое *)
  fb_P_masla_smazki_nizkoe_LA(ai := ai.P_masla_smazki_nizkoe, StrAIp := protections.P_masla_smazki_nizkoe_LA);

  (* Вибрация СТД т.1 *)
  fb_Vibratciia_STD_t1_HA(ai := ai.Vibratciia_STD_t1, StrAIp := protections.Vibratciia_STD_t1_HA);

  (* Вибрация СТД т.2 *)
  fb_Vibratciia_STD_t2_HA(ai := ai.Vibratciia_STD_t2, StrAIp := protections.Vibratciia_STD_t2_HA);

  (* Вибрация ротора нагнетателя т.1 *)
  fb_Vibratciia_rotora_nagnetatelia_t1_HA(ai := ai.Vibratciia_rotora_nagnetatelia_t1, StrAIp := protections.Vibratciia_rotora_nagnetatelia_t1_HA);

  (* Вибрация ротора нагнетателя т.2 *)
  fb_Vibratciia_rotora_nagnetatelia_t2_HA(ai := ai.Vibratciia_rotora_nagnetatelia_t2, StrAIp := protections.Vibratciia_rotora_nagnetatelia_t2_HA);

  (* Вибрация ротора нагнетателя т.3 *)
  fb_Vibratciia_rotora_nagnetatelia_t3_HA(ai := ai.Vibratciia_rotora_nagnetatelia_t3, StrAIp := protections.Vibratciia_rotora_nagnetatelia_t3_HA);

  (* Вибрация ротора нагнетателя т.4 *)
  fb_Vibratciia_rotora_nagnetatelia_t4_HA(ai := ai.Vibratciia_rotora_nagnetatelia_t4, StrAIp := protections.Vibratciia_rotora_nagnetatelia_t4_HA);

  (* Осевой сдвиг ротора нагнетателя *)
  fb_Osevoi_sdvig_rotora_nagnetatelia_HA(ai := ai.Osevoi_sdvig_rotora_nagnetatelia, StrAIp := protections.Osevoi_sdvig_rotora_nagnetatelia_HA);

  (* Уровень масла в маслобаке *)
  fb_Uroven_masla_v_maslobake_LA(ai := ai.Uroven_masla_v_maslobake, StrAIp := protections.Uroven_masla_v_maslobake_LA);
END_FUNCTION_BLOCK

FUNCTION resetDiProtection : BOOL
  VAR_IN_OUT
    protection : struct_DiProtection;
  END_VAR
  VAR CONSTANT
    cmdReset : WORD := 2;
  END_VAR

  IF protection.isRunning THEN
                      protection.inOpcCommandsDisabled:=TRUE;
  		protection.inCommand_Alg:=cmdReset;
  END_IF;
END_FUNCTION

FUNCTION resetAiProtection : BOOL
  VAR_IN_OUT
    protection : struct_AiProtection;
  END_VAR
  VAR CONSTANT
    cmdReset : WORD := 2;
  END_VAR

  IF protection.isRunning THEN
                      protection.inOpcCommandsDisabled:=TRUE;
  		protection.inCommand_Alg:=cmdReset;
  END_IF;
END_FUNCTION

FUNCTION resetAllProtections : BOOL
  VAR_IN_OUT
    protections : ProtectionsConfig;
  END_VAR

  resetAiProtection(protections.T_perednego_opornogo_podshipnika_dvigatelia_t1_HA);
  resetAiProtection(protections.T_zadnego_opornogo_podshipnika_dvigatelia_t2_HA);
  resetAiProtection(protections.T_podshipnika_reduktora_t1_HA);
  resetAiProtection(protections.T_podshipnika_reduktora_t2_HA);
  resetAiProtection(protections.T_podshipnika_reduktora_t3_HA);
  resetAiProtection(protections.T_podshipnika_reduktora_t4_HA);
  resetAiProtection(protections.T_opornogo_podshipnika_nagnetatelia_t1_HA);
  resetAiProtection(protections.T_opornogo_podshipnika_nagnetatelia_t2_HA);
  resetAiProtection(protections.T_opornogo_podshipnika_nagnetatelia_t3_HA);
  resetAiProtection(protections.T_opornoupornogo_podshipnika_nagnetatelia_t4_HA);
  resetAiProtection(protections.T_gaza_na_vykhode_nagnetatelia_HA);
  resetAiProtection(protections.dP_maslogaz_LA);
  resetAiProtection(protections.P_masla_smazki_nizkoe_LA);
  resetAiProtection(protections.Vibratciia_STD_t1_HA);
  resetAiProtection(protections.Vibratciia_STD_t2_HA);
  resetAiProtection(protections.Vibratciia_rotora_nagnetatelia_t1_HA);
  resetAiProtection(protections.Vibratciia_rotora_nagnetatelia_t2_HA);
  resetAiProtection(protections.Vibratciia_rotora_nagnetatelia_t3_HA);
  resetAiProtection(protections.Vibratciia_rotora_nagnetatelia_t4_HA);
  resetAiProtection(protections.Osevoi_sdvig_rotora_nagnetatelia_HA);
  resetAiProtection(protections.Uroven_masla_v_maslobake_LA);
